C01778=1015.719,145.333,-122.552,166.904,54.935,160.108
C01779=1015.715,145.084,-122.532,166.901,54.946,160.110
C01780=1015.710,144.834,-122.514,166.899,54.957,160.111
C01781=1015.706,144.585,-122.494,166.895,54.967,160.113
C01782=1015.702,144.336,-122.475,166.892,54.977,160.114
C01783=1015.696,144.086,-122.456,166.888,54.988,160.115
C01784=1015.692,143.837,-122.437,166.885,54.998,160.116
C01785=1015.687,143.588,-122.418,166.881,55.009,160.118
C01786=1015.683,143.339,-122.399,166.879,55.020,160.119
C01787=1015.678,143.090,-122.380,166.875,55.030,160.121
C01788=1015.674,142.841,-122.360,166.871,55.041,160.122
C01789=1015.669,142.591,-122.342,166.868,55.051,160.123
C01790=1015.665,142.342,-122.323,166.865,55.061,160.125
C01791=1015.661,142.093,-122.303,166.862,55.072,160.126
C01792=1015.655,141.843,-122.285,166.858,55.082,160.127
C01793=1015.651,141.594,-122.265,166.856,55.093,160.129
C01794=1015.647,141.345,-122.247,166.853,55.104,160.130
C01795=1015.642,141.096,-122.228,166.848,55.114,160.131
C01796=1015.637,140.847,-122.208,166.845,55.125,160.133
C01797=1015.633,140.597,-122.189,166.842,55.135,160.134
C01798=1015.628,140.348,-122.171,166.839,55.145,160.136
C01799=1015.624,140.099,-122.152,166.836,55.156,160.137
C01800=1015.619,139.850,-122.133,166.832,55.166,160.138
C01801=1015.615,139.601,-122.113,166.829,55.176,160.140
C01802=1015.611,139.351,-122.095,166.827,55.188,160.141
C01803=1015.606,139.106,-122.076,166.823,55.197,160.142
C01804=1015.602,138.863,-122.057,166.820,55.208,160.144
C01805=1015.598,138.618,-122.039,166.817,55.218,160.145
C01806=1015.594,138.374,-122.021,166.813,55.228,160.146
C01807=1015.588,138.130,-122.002,166.810,55.239,160.148
C01808=1015.584,137.886,-121.984,166.807,55.249,160.149
C01809=1015.580,137.641,-121.965,166.804,55.259,160.150
C01810=1015.575,137.397,-121.946,166.801,55.270,160.152
C01811=1015.571,137.147,-121.927,166.798,55.280,160.153
C01812=1015.566,136.898,-121.909,166.795,55.291,160.155
C01813=1015.561,136.649,-121.890,166.791,55.301,160.156
C01814=1015.557,136.400,-121.872,166.788,55.311,160.157
C01815=1015.552,136.151,-121.853,166.785,55.322,160.159
C01816=1015.548,135.901,-121.834,166.781,55.332,160.160
C01817=1015.543,135.652,-121.816,166.778,55.344,160.161
C01818=1015.539,135.403,-121.796,166.775,55.354,160.163
C01819=1015.534,135.153,-121.778,166.772,55.364,160.164
C01820=1015.530,134.904,-121.759,166.769,55.375,160.165
C01821=1015.525,134.655,-121.740,166.766,55.385,160.167
C01822=1015.521,134.406,-121.723,166.763,55.396,160.168
C01823=1015.517,134.157,-121.704,166.760,55.406,160.170
C01824=1015.512,133.907,-121.686,166.757,55.417,160.171
C01825=1015.507,133.658,-121.666,166.753,55.428,160.172
C01826=1015.503,133.409,-121.648,166.750,55.438,160.174
C01827=1015.498,133.160,-121.630,166.747,55.449,160.175
C01828=1015.493,132.911,-121.610,166.744,55.459,160.176
C01829=1015.489,132.661,-121.592,166.741,55.470,160.178
C01830=1015.485,132.412,-121.574,166.737,55.480,160.179
C01831=1015.479,132.121,-121.552,166.734,55.492,160.181
C01832=1015.474,131.830,-121.531,166.730,55.505,160.183
C01833=1015.469,131.539,-121.509,166.727,55.517,160.184
C01834=1015.463,131.249,-121.487,166.723,55.529,160.186
C01835=1015.459,131.000,-121.469,166.719,55.540,160.187
C01836=1015.454,130.750,-121.451,166.717,55.551,160.189
C01837=1015.450,130.501,-121.432,166.714,55.561,160.190
C01838=1015.446,130.252,-121.414,166.711,55.572,160.191
C01839=1015.441,130.003,-121.395,166.708,55.582,160.193
C01840=1015.437,129.753,-121.376,166.705,55.592,160.194
C01841=1015.432,129.504,-121.358,166.702,55.603,160.195
C01842=1015.427,129.255,-121.340,166.698,55.613,160.197
C01843=1015.423,129.005,-121.321,166.695,55.624,160.198
C01844=1015.418,128.756,-121.303,166.693,55.635,160.200
C01845=1015.413,128.506,-121.285,166.690,55.645,160.201
C01846=1015.409,128.257,-121.267,166.687,55.656,160.203
C01847=1015.404,128.008,-121.249,166.683,55.667,160.204
C01848=1015.400,127.759,-121.231,166.680,55.677,160.205
C01849=1015.395,127.510,-121.213,166.677,55.688,160.207
C01850=1015.390,127.260,-121.195,166.674,55.699,160.208
C01851=1015.386,127.010,-121.177,166.671,55.709,160.210
C01852=1015.381,126.761,-121.159,166.668,55.720,160.211
C01853=1015.376,126.512,-121.141,166.666,55.731,160.213
C01854=1015.371,126.262,-121.123,166.663,55.741,160.214
C01855=1015.367,126.014,-121.105,166.658,55.752,160.215
C01856=1015.362,125.764,-121.087,166.655,55.763,160.217
C01857=1015.358,125.515,-121.068,166.652,55.773,160.218
C01858=1015.353,125.266,-121.050,166.649,55.783,160.219
C01859=1015.348,125.016,-121.032,166.647,55.795,160.221
C01860=1015.344,124.767,-121.015,166.644,55.805,160.222
C01861=1015.339,124.518,-120.997,166.641,55.816,160.224
C01862=1015.335,124.268,-120.979,166.638,55.826,160.225
C01863=1015.330,124.019,-120.961,166.635,55.837,160.226
C01864=1015.325,123.770,-120.942,166.632,55.847,160.228
C01865=1015.321,123.521,-120.925,166.629,55.857,160.229
C01866=1015.316,123.271,-120.907,166.626,55.869,160.231
C01867=1015.311,122.990,-120.887,166.623,55.880,160.232
C01868=1015.306,122.709,-120.866,166.619,55.892,160.234
C01869=1015.301,122.429,-120.846,166.617,55.904,160.236
C01870=1015.296,122.148,-120.825,166.612,55.916,160.237
C01871=1015.291,121.899,-120.808,166.609,55.927,160.238
C01872=1015.287,121.650,-120.789,166.606,55.937,160.240
C01873=1015.282,121.400,-120.772,166.603,55.948,160.241
C01874=1015.277,121.150,-120.754,166.600,55.958,160.242
C01875=1015.273,120.902,-120.736,166.597,55.969,160.244
C01876=1015.268,120.652,-120.718,166.594,55.979,160.245
C01877=1015.264,120.402,-120.700,166.591,55.990,160.247
C01878=1015.260,120.154,-120.683,166.589,56.001,160.248
C01879=1015.255,119.904,-120.664,166.587,56.011,160.250
C01880=1015.250,119.655,-120.646,166.584,56.022,160.251
C01881=1015.246,119.405,-120.629,166.581,56.032,160.253
C01882=1015.242,119.156,-120.611,166.578,56.043,160.254
C01883=1015.237,118.907,-120.593,166.575,56.053,160.255
C01884=1015.232,118.658,-120.575,166.572,56.064,160.257
C01885=1015.228,118.408,-120.558,166.569,56.074,160.258
C01886=1015.223,118.159,-120.540,166.566,56.085,160.260
C01887=1015.219,117.910,-120.521,166.563,56.095,160.261
C01888=1015.214,117.660,-120.504,166.560,56.106,160.262
C01889=1015.210,117.411,-120.486,166.557,56.116,160.264
C01890=1015.205,117.162,-120.468,166.555,56.127,160.265
C01891=1015.200,116.912,-120.450,166.551,56.137,160.266
C01892=1015.196,116.663,-120.433,166.548,56.147,160.268
C01893=1015.192,116.414,-120.415,166.545,56.158,160.269
C01894=1015.187,116.164,-120.396,166.542,56.168,160.271
C01895=1015.183,115.915,-120.379,166.540,56.178,160.272
C01896=1015.178,115.666,-120.361,166.538,56.189,160.274
C01897=1015.174,115.417,-120.344,166.535,56.199,160.275
C01898=1015.170,115.167,-120.326,166.532,56.210,160.276
C01899=1015.165,114.918,-120.308,166.529,56.220,160.278
C01900=1015.161,114.669,-120.291,166.526,56.231,160.279
C01901=1015.156,114.419,-120.273,166.523,56.242,160.281
C01902=1015.151,114.170,-120.254,166.520,56.252,160.282
C01903=1015.147,113.921,-120.237,166.518,56.262,160.283
C01904=1015.143,113.671,-120.219,166.515,56.272,160.285
C01905=1015.139,113.422,-120.202,166.512,56.283,160.286
C01906=1015.134,113.173,-120.184,166.509,56.293,160.287
C01907=1015.129,112.923,-120.166,166.506,56.304,160.289
C01908=1015.125,112.674,-120.149,166.503,56.314,160.290
C01909=1015.121,112.425,-120.130,166.500,56.325,160.292
C01910=1015.117,112.175,-120.113,166.498,56.334,160.293
C01911=1015.112,111.926,-120.095,166.495,56.345,160.294
C01912=1015.107,111.676,-120.078,166.492,56.355,160.296
C01913=1015.103,111.427,-120.060,166.490,56.366,160.297
C01914=1015.098,111.178,-120.043,166.487,56.377,160.299
C01915=1015.094,110.928,-120.026,166.484,56.387,160.300
C01916=1015.089,110.679,-120.008,166.481,56.398,160.301
C01917=1015.085,110.429,-119.990,166.478,56.408,160.303
C01918=1015.080,110.181,-119.973,166.475,56.419,160.304
C01919=1015.076,109.931,-119.956,166.472,56.429,160.306
C01920=1015.072,109.682,-119.939,166.471,56.440,160.307
C01921=1015.066,109.433,-119.921,166.468,56.450,160.309
C01922=1015.062,109.183,-119.904,166.465,56.461,160.310
C01923=1015.058,108.933,-119.887,166.462,56.471,160.312
C01924=1015.053,108.684,-119.870,166.459,56.482,160.313
C01925=1015.048,108.435,-119.852,166.456,56.492,160.314
C01926=1015.043,108.185,-119.835,166.454,56.503,160.316
C01927=1015.039,107.936,-119.818,166.451,56.514,160.317
C01928=1015.034,107.686,-119.801,166.448,56.524,160.319
C01929=1015.030,107.438,-119.783,166.445,56.535,160.320
C01930=1015.025,107.188,-119.767,166.442,56.545,160.321
C01931=1015.020,106.907,-119.747,166.439,56.557,160.323
C01932=1015.015,106.626,-119.728,166.436,56.569,160.325
C01933=1015.009,106.346,-119.708,166.434,56.581,160.327
C01934=1015.004,106.065,-119.689,166.431,56.593,160.328
C01935=1015.000,105.816,-119.672,166.428,56.603,160.329
C01936=1014.995,105.566,-119.655,166.425,56.614,160.331
C01937=1014.991,105.317,-119.638,166.422,56.625,160.332
C01938=1014.985,105.068,-119.621,166.419,56.634,160.333
C01939=1014.982,104.819,-119.604,166.416,56.645,160.335
C01940=1014.977,104.569,-119.586,166.413,56.656,160.336
C01941=1014.972,104.320,-119.570,166.411,56.666,160.338
C01942=1014.968,104.070,-119.552,166.409,56.676,160.339
C01943=1014.963,103.821,-119.536,166.406,56.687,160.341
C01944=1014.959,103.571,-119.518,166.403,56.698,160.342
C01945=1014.954,103.323,-119.501,166.401,56.708,160.344
C01946=1014.950,103.073,-119.484,166.398,56.719,160.345
C01947=1014.945,102.824,-119.467,166.395,56.729,160.346
C01948=1014.941,102.574,-119.450,166.392,56.740,160.348
C01949=1014.936,102.325,-119.433,166.390,56.750,160.349
C01950=1014.932,102.075,-119.416,166.387,56.760,160.351
C01951=1014.927,101.826,-119.399,166.385,56.771,160.352
C01952=1014.923,101.576,-119.382,166.382,56.782,160.354
C01953=1014.918,101.327,-119.366,166.378,56.792,160.355
C01954=1014.914,101.078,-119.348,166.377,56.802,160.356
C01955=1014.909,100.829,-119.332,166.374,56.812,160.358
C01956=1014.905,100.579,-119.315,166.371,56.823,160.359
C01957=1014.900,100.330,-119.298,166.368,56.833,160.360
C01958=1014.895,100.080,-119.280,166.365,56.844,160.362
C01959=1014.891,99.831,-119.263,166.364,56.854,160.363
C01960=1014.886,99.581,-119.246,166.361,56.864,160.365
C01961=1014.882,99.332,-119.229,166.358,56.874,160.366
C01962=1014.878,99.083,-119.212,166.355,56.885,160.367
C01963=1014.872,98.833,-119.196,166.353,56.895,160.369
C01964=1014.869,98.584,-119.179,166.350,56.906,160.370
C01965=1014.864,98.334,-119.162,166.348,56.917,160.372
C01966=1014.859,98.085,-119.146,166.345,56.927,160.373
C01967=1014.854,97.836,-119.129,166.342,56.938,160.375
C01968=1014.849,97.586,-119.112,166.339,56.948,160.376
C01969=1014.845,97.337,-119.095,166.336,56.959,160.377
C01970=1014.840,97.087,-119.079,166.335,56.969,160.379
C01971=1014.836,96.838,-119.063,166.332,56.979,160.381
C01972=1014.831,96.589,-119.046,166.329,56.990,160.382
C01973=1014.827,96.339,-119.029,166.327,57.001,160.383
C01974=1014.822,96.090,-119.012,166.323,57.011,160.385
C01975=1014.818,95.841,-118.996,166.321,57.021,160.386
C01976=1014.813,95.591,-118.980,166.319,57.032,160.388
C01977=1014.808,95.342,-118.963,166.316,57.042,160.389
C01978=1014.804,95.092,-118.946,166.314,57.053,160.391
C01979=1014.799,94.843,-118.929,166.310,57.063,160.392
C01980=1014.795,94.593,-118.914,166.308,57.074,160.393
C01981=1014.789,94.344,-118.897,166.306,57.084,160.395
C01982=1014.785,94.095,-118.880,166.303,57.095,160.396
C01983=1014.781,93.845,-118.863,166.300,57.105,160.397
C01984=1014.776,93.595,-118.847,166.298,57.115,160.399
C01985=1014.771,93.346,-118.831,166.296,57.126,160.401
C01986=1014.767,93.097,-118.814,166.293,57.136,160.402
C01987=1014.762,92.847,-118.797,166.290,57.146,160.403
C01988=1014.758,92.598,-118.781,166.287,57.157,160.405
C01989=1014.753,92.349,-118.764,166.286,57.167,160.406
C01990=1014.749,92.100,-118.748,166.283,57.177,160.407
C01991=1014.744,91.850,-118.731,166.280,57.188,160.409
C01992=1014.740,91.600,-118.715,166.277,57.199,160.410
C01993=1014.735,91.351,-118.698,166.275,57.208,160.412
C01994=1014.730,91.102,-118.681,166.273,57.219,160.413
C01995=1014.725,90.821,-118.663,166.269,57.231,160.415
C01996=1014.721,90.541,-118.645,166.267,57.242,160.416
C01997=1014.715,90.260,-118.626,166.264,57.254,160.418
C01998=1014.710,89.980,-118.608,166.261,57.265,160.419
C01999=1014.705,89.730,-118.591,166.259,57.275,160.421
C02000=1014.701,89.481,-118.574,166.256,57.286,160.422
C02001=1014.697,89.232,-118.558,166.253,57.296,160.424
C02002=1014.692,88.983,-118.542,166.252,57.306,160.425
C02003=1014.687,88.732,-118.526,166.249,57.316,160.426
C02004=1014.683,88.483,-118.509,166.246,57.327,160.428
C02005=1014.678,88.234,-118.493,166.243,57.338,160.429
C02006=1014.674,87.985,-118.477,166.241,57.347,160.431
C02007=1014.669,87.735,-118.461,166.239,57.358,160.432
C02008=1014.664,87.486,-118.444,166.236,57.369,160.434
C02009=1014.660,87.236,-118.428,166.233,57.380,160.435
C02010=1014.655,86.987,-118.412,166.231,57.389,160.437
C02011=1014.650,86.737,-118.396,166.229,57.400,160.438
C02012=1014.645,86.488,-118.380,166.226,57.411,160.439
C02013=1014.641,86.239,-118.364,166.223,57.421,160.441
C02014=1014.637,85.989,-118.348,166.222,57.431,160.442
C02015=1014.631,85.739,-118.332,166.219,57.442,160.444
C02016=1014.627,85.490,-118.316,166.216,57.452,160.445
C02017=1014.622,85.241,-118.299,166.213,57.463,160.446
C02018=1014.618,84.991,-118.284,166.212,57.473,160.448
C02019=1014.614,84.742,-118.268,166.209,57.483,160.449
C02020=1014.608,84.492,-118.252,166.206,57.494,160.451
C02021=1014.604,84.243,-118.236,166.204,57.503,160.452
C02022=1014.599,83.994,-118.219,166.201,57.514,160.454
C02023=1014.595,83.744,-118.203,166.199,57.525,160.455
C02024=1014.590,83.495,-118.188,166.197,57.534,160.456
C02025=1014.586,83.246,-118.171,166.194,57.545,160.458
C02026=1014.581,82.995,-118.155,166.191,57.555,160.459
C02027=1014.577,82.746,-118.139,166.189,57.566,160.461
C02028=1014.571,82.497,-118.123,166.186,57.575,160.462
C02029=1014.567,82.248,-118.108,166.184,57.586,160.464
C02030=1014.563,81.998,-118.092,166.182,57.596,160.465
C02031=1014.558,81.749,-118.075,166.179,57.607,160.466
C02032=1014.553,81.499,-118.059,166.176,57.617,160.468
C02033=1014.549,81.249,-118.044,166.175,57.627,160.469
C02034=1014.544,81.000,-118.027,166.172,57.637,160.470
C02035=1014.540,80.751,-118.011,166.169,57.648,160.472
C02036=1014.535,80.501,-117.995,166.167,57.657,160.473
C02037=1014.530,80.252,-117.980,166.165,57.668,160.475
C02038=1014.526,80.003,-117.964,166.163,57.678,160.476
C02039=1014.521,79.753,-117.948,166.159,57.688,160.477
C02040=1014.517,79.503,-117.932,166.157,57.699,160.479
C02041=1014.512,79.254,-117.915,166.155,57.708,160.480
C02042=1014.508,79.004,-117.900,166.152,57.719,160.482
C02043=1014.503,78.755,-117.884,166.150,57.729,160.483
C02044=1014.499,78.506,-117.867,166.147,57.739,160.484
C02045=1014.494,78.257,-117.852,166.146,57.749,160.486
C02046=1014.489,78.007,-117.836,166.143,57.759,160.487
C02047=1014.485,77.758,-117.821,166.141,57.769,160.489
C02048=1014.480,77.508,-117.804,166.138,57.780,160.490
C02049=1014.476,77.258,-117.788,166.135,57.790,160.491
C02050=1014.471,77.009,-117.772,166.133,57.799,160.493
C02051=1014.467,76.759,-117.757,166.131,57.810,160.494
C02052=1014.462,76.510,-117.741,166.129,57.820,160.496
C02053=1014.458,76.260,-117.726,166.126,57.831,160.497
C02054=1014.453,76.011,-117.709,166.124,57.840,160.499
C02055=1014.448,75.762,-117.694,166.121,57.850,160.500
C02056=1014.444,75.513,-117.678,166.119,57.861,160.501
C02057=1014.439,75.263,-117.662,166.117,57.871,160.503
C02058=1014.434,75.014,-117.647,166.114,57.882,160.504
C02059=1014.429,74.733,-117.630,166.112,57.892,160.506
C02060=1014.424,74.453,-117.613,166.109,57.904,160.507
C02061=1014.419,74.173,-117.595,166.107,57.915,160.509
C02062=1014.413,73.893,-117.577,166.104,57.927,160.510
C02063=1014.409,73.643,-117.562,166.102,57.937,160.512
C02064=1014.404,73.394,-117.546,166.099,57.947,160.513
C02065=1014.400,73.144,-117.531,166.096,57.958,160.514
C02066=1014.395,72.895,-117.515,166.094,57.967,160.516
C02067=1014.390,72.645,-117.500,166.091,57.978,160.517
C02068=1014.386,72.396,-117.484,166.090,57.988,160.519
C02069=1014.380,72.146,-117.468,166.087,57.998,160.520
C02070=1014.376,71.896,-117.453,166.085,58.008,160.521
C02071=1014.372,71.647,-117.437,166.083,58.019,160.523
C02072=1014.367,71.397,-117.422,166.081,58.028,160.524
C02073=1014.363,71.148,-117.406,166.078,58.038,160.526
C02074=1014.357,70.899,-117.391,166.076,58.048,160.527
C02075=1014.353,70.649,-117.375,166.073,58.059,160.529
C02076=1014.348,70.399,-117.361,166.071,58.068,160.530
C02077=1014.344,70.150,-117.345,166.068,58.079,160.531
C02078=1014.340,69.900,-117.329,166.066,58.088,160.533
C02079=1014.335,69.651,-117.314,166.063,58.098,160.534
C02080=1014.331,69.402,-117.298,166.062,58.109,160.535
C02081=1014.326,69.153,-117.283,166.059,58.119,160.537
C02082=1014.322,68.903,-117.267,166.057,58.129,160.538
C02083=1014.317,68.654,-117.252,166.054,58.139,160.539
C02084=1014.312,68.404,-117.237,166.052,58.148,160.541
C02085=1014.307,68.155,-117.221,166.050,58.159,160.542
C02086=1014.303,67.905,-117.206,166.048,58.169,160.544
C02087=1014.298,67.655,-117.191,166.046,58.179,160.545
C02088=1014.294,67.406,-117.175,166.043,58.189,160.546
C02089=1014.289,67.157,-117.160,166.041,58.198,160.548
C02090=1014.284,66.907,-117.145,166.038,58.209,160.549
C02091=1014.280,66.657,-117.130,166.037,58.219,160.551
C02092=1014.275,66.408,-117.115,166.034,58.229,160.552
C02093=1014.271,66.158,-117.099,166.032,58.239,160.553
C02094=1014.265,65.909,-117.084,166.029,58.249,160.555
C02095=1014.261,65.659,-117.069,166.027,58.259,160.556
C02096=1014.256,65.410,-117.054,166.024,58.269,160.557
C02097=1014.251,65.160,-117.038,166.022,58.279,160.559
C02098=1014.247,64.910,-117.023,166.020,58.289,160.560
C02099=1014.243,64.662,-117.009,166.018,58.299,160.562
C02100=1014.238,64.412,-116.993,166.016,58.309,160.563
C02101=1014.234,64.163,-116.978,166.013,58.319,160.564
C02102=1014.229,63.913,-116.963,166.011,58.329,160.566
C02103=1014.224,63.664,-116.948,166.008,58.339,160.567
C02104=1014.220,63.414,-116.932,166.007,58.349,160.568
C02105=1014.215,63.164,-116.918,166.004,58.359,160.570
C02106=1014.210,62.915,-116.903,166.002,58.368,160.571
C02107=1014.206,62.665,-116.888,166.000,58.378,160.572
C02108=1014.201,62.415,-116.872,165.997,58.388,160.574
C02109=1014.196,62.167,-116.858,165.995,58.398,160.575
C02110=1014.192,61.917,-116.843,165.993,58.409,160.577
C02111=1014.187,61.667,-116.829,165.991,58.419,160.578
C02112=1014.182,61.418,-116.813,165.988,58.429,160.579
C02113=1014.177,61.168,-116.799,165.986,58.439,160.581
C02114=1014.172,60.919,-116.784,165.983,58.449,160.582
C02115=1014.167,60.669,-116.769,165.981,58.458,160.583
C02116=1014.162,60.419,-116.754,165.979,58.469,160.585
C02117=1014.158,60.170,-116.740,165.977,58.479,160.586
C02118=1014.153,59.921,-116.725,165.974,58.489,160.588
C02119=1014.148,59.671,-116.710,165.973,58.499,160.589
C02120=1014.144,59.421,-116.696,165.970,58.509,160.590
C02121=1014.138,59.172,-116.681,165.968,58.519,160.592
C02122=1014.134,58.922,-116.666,165.966,58.529,160.593
C02123=1014.129,58.642,-116.649,165.963,58.540,160.595
C02124=1014.123,58.362,-116.633,165.961,58.551,160.596
C02125=1014.118,58.082,-116.617,165.958,58.562,160.598
C02126=1014.113,57.802,-116.600,165.955,58.573,160.599
C02127=1014.108,57.552,-116.585,165.953,58.583,160.600
C02128=1014.103,57.303,-116.570,165.951,58.593,160.602
C02129=1014.099,57.053,-116.556,165.948,58.603,160.603
C02130=1014.094,56.804,-116.542,165.947,58.613,160.605
C02131=1014.089,56.554,-116.527,165.944,58.623,160.606
C02132=1014.085,56.304,-116.512,165.942,58.633,160.607
C02133=1014.080,56.055,-116.498,165.940,58.642,160.609
C02134=1014.075,55.805,-116.482,165.937,58.653,160.610
C02135=1014.071,55.556,-116.468,165.936,58.662,160.611
C02136=1014.066,55.306,-116.454,165.934,58.672,160.613
C02137=1014.061,55.057,-116.439,165.931,58.682,160.614
C02138=1014.056,54.807,-116.424,165.928,58.691,160.615
C02139=1014.052,54.558,-116.410,165.927,58.701,160.617
C02140=1014.047,54.309,-116.395,165.924,58.711,160.618
C02141=1014.042,54.059,-116.381,165.922,58.721,160.619
C02142=1014.038,53.809,-116.366,165.920,58.731,160.621
C02143=1014.033,53.560,-116.351,165.918,58.740,160.622
C02144=1014.028,53.310,-116.337,165.915,58.750,160.623
C02145=1014.024,53.061,-116.322,165.913,58.760,160.625
C02146=1014.019,52.811,-116.307,165.912,58.770,160.626
C02147=1014.015,52.562,-116.293,165.910,58.779,160.628
C02148=1014.010,52.312,-116.279,165.906,58.789,160.629
C02149=1014.005,52.062,-116.264,165.905,58.799,160.630
C02150=1014.000,51.813,-116.249,165.903,58.808,160.632
C02151=1013.996,51.564,-116.235,165.900,58.817,160.633
C02152=1013.991,51.314,-116.220,165.898,58.828,160.634
C02153=1013.986,51.064,-116.206,165.896,58.837,160.635
C02154=1013.982,50.816,-116.191,165.894,58.847,160.637
C02155=1013.977,50.566,-116.177,165.892,58.856,160.638
C02156=1013.972,50.316,-116.162,165.890,58.866,160.640
C02157=1013.968,50.066,-116.148,165.888,58.875,160.641
C02158=1013.963,49.817,-116.133,165.885,58.885,160.642
C02159=1013.959,49.567,-116.119,165.883,58.894,160.643
C02160=1013.954,49.318,-116.104,165.881,58.904,160.645
C02161=1013.950,49.068,-116.090,165.878,58.913,160.646
C02162=1013.945,48.818,-116.076,165.877,58.923,160.647
C02163=1013.940,48.569,-116.060,165.875,58.933,160.649
C02164=1013.936,48.320,-116.046,165.873,58.942,160.650
C02165=1013.931,48.070,-116.032,165.870,58.952,160.651
C02166=1013.926,47.820,-116.017,165.868,58.961,160.652
C02167=1013.922,47.571,-116.003,165.866,58.971,160.654
C02168=1013.917,47.322,-115.988,165.863,58.980,160.655
C02169=1013.912,47.072,-115.974,165.861,58.989,160.656
C02170=1013.908,46.823,-115.960,165.859,58.999,160.657
C02171=1013.903,46.573,-115.945,165.857,59.008,160.659
C02172=1013.899,46.323,-115.931,165.855,59.018,160.660
C02173=1013.895,46.074,-115.917,165.853,59.027,160.661
C02174=1013.890,45.824,-115.901,165.851,59.036,160.662
C02175=1013.885,45.575,-115.887,165.849,59.046,160.664
C02176=1013.881,45.325,-115.873,165.847,59.055,160.665
C02177=1013.876,45.076,-115.858,165.845,59.065,160.667
C02178=1013.872,44.826,-115.844,165.843,59.074,160.668
C02179=1013.867,44.576,-115.830,165.840,59.083,160.669
C02180=1013.862,44.327,-115.815,165.839,59.093,160.670
C02181=1013.858,44.078,-115.801,165.836,59.102,160.671
C02182=1013.853,43.828,-115.786,165.834,59.111,160.673
C02183=1013.849,43.579,-115.772,165.832,59.120,160.674
C02184=1013.844,43.329,-115.758,165.830,59.130,160.675
C02185=1013.840,43.079,-115.743,165.828,59.139,160.676
C02186=1013.835,42.830,-115.729,165.825,59.148,160.678
C02187=1013.830,42.549,-115.713,165.823,59.158,160.679
C02188=1013.825,42.270,-115.696,165.821,59.169,160.680
C02189=1013.820,41.990,-115.680,165.819,59.179,160.682
C02190=1013.815,41.709,-115.665,165.816,59.189,160.683
C02191=1013.811,41.460,-115.650,165.814,59.198,160.684
C02192=1013.805,41.210,-115.637,165.812,59.208,160.686
C02193=1013.801,40.961,-115.622,165.810,59.217,160.687
C02194=1013.796,40.711,-115.608,165.808,59.226,160.688
C02195=1013.792,40.461,-115.595,165.806,59.236,160.690
C02196=1013.787,40.212,-115.581,165.804,59.245,160.691
C02197=1013.782,39.962,-115.566,165.802,59.254,160.692
C02198=1013.778,39.713,-115.552,165.799,59.263,160.693
C02199=1013.773,39.463,-115.538,165.798,59.273,160.695
C02200=1013.768,39.214,-115.524,165.795,59.282,160.696
C02201=1013.764,38.964,-115.510,165.793,59.292,160.697
C02202=1013.760,38.715,-115.496,165.791,59.301,160.698
C02203=1013.754,38.465,-115.483,165.789,59.310,160.699
C02204=1013.750,38.215,-115.468,165.787,59.320,160.701
C02205=1013.745,37.965,-115.454,165.785,59.329,160.702
C02206=1013.741,37.717,-115.441,165.782,59.338,160.703
C02207=1013.736,37.467,-115.426,165.780,59.347,160.704
C02208=1013.732,37.218,-115.412,165.778,59.356,160.706
C02209=1013.727,36.967,-115.399,165.776,59.365,160.707
C02210=1013.722,36.718,-115.385,165.774,59.374,160.708
C02211=1013.718,36.468,-115.370,165.772,59.383,160.709
C02212=1013.713,36.218,-115.356,165.770,59.392,160.710
C02213=1013.708,35.969,-115.343,165.768,59.401,160.712
C02214=1013.704,35.719,-115.329,165.766,59.411,160.713
C02215=1013.699,35.470,-115.315,165.764,59.420,160.714
C02216=1013.694,35.220,-115.302,165.762,59.429,160.716
C02217=1013.689,34.971,-115.288,165.759,59.438,160.717
C02218=1013.685,34.722,-115.274,165.757,59.447,160.718
C02219=1013.680,34.471,-115.261,165.755,59.457,160.719
C02220=1013.675,34.223,-115.247,165.753,59.466,160.720
C02221=1013.671,33.972,-115.233,165.750,59.475,160.721
C02222=1013.666,33.723,-115.220,165.749,59.484,160.723
C02223=1013.661,33.473,-115.205,165.748,59.493,160.724
C02224=1013.657,33.224,-115.193,165.745,59.502,160.726
C02225=1013.652,32.974,-115.178,165.743,59.512,160.727
C02226=1013.647,32.724,-115.165,165.741,59.521,160.728
C02227=1013.642,32.475,-115.151,165.739,59.530,160.729
C02228=1013.638,32.226,-115.137,165.737,59.539,160.730
C02229=1013.633,31.976,-115.125,165.735,59.547,160.731
C02230=1013.628,31.726,-115.110,165.733,59.556,160.732
C02231=1013.624,31.477,-115.097,165.730,59.565,160.734
C02232=1013.619,31.227,-115.083,165.728,59.574,160.735
C02233=1013.615,30.977,-115.070,165.726,59.584,160.736
C02234=1013.610,30.727,-115.056,165.725,59.592,160.737
C02235=1013.605,30.478,-115.043,165.723,59.601,160.739
C02236=1013.600,30.229,-115.029,165.720,59.610,160.740
C02237=1013.596,29.979,-115.015,165.718,59.620,160.741
C02238=1013.591,29.730,-115.002,165.716,59.628,160.742
C02239=1013.586,29.480,-114.988,165.714,59.637,160.743
C02240=1013.582,29.230,-114.975,165.712,59.646,160.744
C02241=1013.578,28.981,-114.961,165.710,59.655,160.746
C02242=1013.572,28.731,-114.948,165.709,59.664,160.747
C02243=1013.568,28.482,-114.934,165.706,59.672,160.748
C02244=1013.563,28.232,-114.920,165.704,59.681,160.749
C02245=1013.558,27.983,-114.907,165.703,59.690,160.750
C02246=1013.554,27.733,-114.894,165.700,59.698,160.751
C02247=1013.549,27.483,-114.880,165.698,59.708,160.753
C02248=1013.545,27.234,-114.866,165.696,59.716,160.754
C02249=1013.540,26.983,-114.853,165.694,59.725,160.755
C02250=1013.535,26.734,-114.840,165.691,59.734,160.756
C02251=1013.530,26.454,-114.825,165.690,59.744,160.758
C02252=1013.525,26.174,-114.810,165.687,59.754,160.759
C02253=1013.520,25.894,-114.794,165.685,59.763,160.760
C02254=1013.515,25.615,-114.780,165.683,59.774,160.761
C02255=1013.509,25.365,-114.766,165.680,59.783,160.763
C02256=1013.505,25.115,-114.754,165.679,59.791,160.764
C02257=1013.501,24.866,-114.740,165.677,59.800,160.765
C02258=1013.496,24.616,-114.726,165.674,59.809,160.766
C02259=1013.491,24.367,-114.714,165.673,59.817,160.767
C02260=1013.486,24.117,-114.701,165.670,59.826,160.768
C02261=1013.481,23.867,-114.688,165.668,59.835,160.769
C02262=1013.477,23.618,-114.674,165.667,59.843,160.771
C02263=1013.473,23.368,-114.661,165.664,59.853,160.772
C02264=1013.467,23.118,-114.648,165.662,59.861,160.773
C02265=1013.462,22.869,-114.634,165.661,59.870,160.774
C02266=1013.458,22.620,-114.621,165.658,59.878,160.775
C02267=1013.453,22.369,-114.608,165.657,59.887,160.776
C02268=1013.449,22.120,-114.595,165.654,59.895,160.777
C02269=1013.444,21.870,-114.582,165.653,59.904,160.779
C02270=1013.439,21.621,-114.569,165.650,59.912,160.779
C02271=1013.434,21.371,-114.555,165.648,59.922,160.781
C02272=1013.430,21.122,-114.543,165.646,59.930,160.782
C02273=1013.426,20.872,-114.529,165.644,59.939,160.783
C02274=1013.421,20.623,-114.516,165.642,59.947,160.784
C02275=1013.416,20.373,-114.503,165.639,59.955,160.785
C02276=1013.411,20.123,-114.490,165.638,59.964,160.786
C02277=1013.407,19.874,-114.477,165.636,59.972,160.787
C02278=1013.402,19.623,-114.463,165.635,59.981,160.789
C02279=1013.397,19.374,-114.450,165.632,59.990,160.790
C02280=1013.393,19.125,-114.437,165.630,59.998,160.791
C02281=1013.388,18.875,-114.424,165.628,60.007,160.792
C02282=1013.383,18.625,-114.411,165.626,60.015,160.793
C02283=1013.379,18.376,-114.398,165.623,60.023,160.794
C02284=1013.374,18.126,-114.386,165.622,60.032,160.795
C02285=1013.370,17.876,-114.372,165.620,60.040,160.796
C02286=1013.365,17.626,-114.359,165.618,60.048,160.797
C02287=1013.360,17.377,-114.346,165.615,60.057,160.798
C02288=1013.356,17.127,-114.333,165.614,60.066,160.799
C02289=1013.351,16.878,-114.321,165.612,60.074,160.801
C02290=1013.347,16.628,-114.308,165.610,60.082,160.801
C02291=1013.342,16.378,-114.295,165.608,60.090,160.802
C02292=1013.337,16.129,-114.282,165.606,60.099,160.804
C02293=1013.332,15.880,-114.268,165.604,60.107,160.805
C02294=1013.328,15.630,-114.256,165.601,60.116,160.806
C02295=1013.323,15.381,-114.243,165.600,60.124,160.807
C02296=1013.318,15.131,-114.230,165.598,60.132,160.808
C02297=1013.313,14.881,-114.217,165.596,60.141,160.809
C02298=1013.309,14.632,-114.204,165.594,60.149,160.810
C02299=1013.304,14.382,-114.191,165.593,60.157,160.811
C02300=1013.300,14.133,-114.179,165.590,60.165,160.812
C02301=1013.295,13.883,-114.166,165.588,60.173,160.813
C02302=1013.290,13.633,-114.153,165.587,60.181,160.814
C02303=1013.286,13.383,-114.141,165.584,60.190,160.815
C02304=1013.281,13.133,-114.128,165.582,60.198,160.816
C02305=1013.276,12.884,-114.115,165.580,60.206,160.817
C02306=1013.272,12.634,-114.102,165.578,60.214,160.818
C02307=1013.267,12.384,-114.089,165.576,60.222,160.819
C02308=1013.261,12.135,-114.077,165.574,60.230,160.820
C02309=1013.257,11.885,-114.065,165.572,60.240,160.822
C02310=1013.252,11.635,-114.052,165.571,60.248,160.823
C02311=1013.248,11.386,-114.039,165.568,60.256,160.824
C02312=1013.243,11.137,-114.027,165.566,60.264,160.825
C02313=1013.238,10.887,-114.014,165.565,60.272,160.826
C02314=1013.234,10.637,-114.002,165.562,60.281,160.827
C02315=1013.228,10.358,-113.988,165.560,60.290,160.828
C02316=1013.223,10.080,-113.975,165.557,60.298,160.829
C02317=1013.218,9.801,-113.960,165.555,60.308,160.830
C02318=1013.212,9.523,-113.946,165.553,60.317,160.831
C02319=1013.208,9.274,-113.933,165.551,60.325,160.832
C02320=1013.203,9.024,-113.922,165.550,60.333,160.833
C02321=1013.198,8.774,-113.909,165.548,60.341,160.835
C02322=1013.193,8.524,-113.896,165.545,60.349,160.835
C02323=1013.189,8.274,-113.884,165.543,60.357,160.836
C02324=1013.183,8.025,-113.872,165.541,60.365,160.837
C02325=1013.179,7.776,-113.859,165.540,60.373,160.838
C02326=1013.174,7.526,-113.846,165.538,60.381,160.840
C02327=1013.170,7.276,-113.834,165.535,60.389,160.840
C02328=1013.165,7.027,-113.822,165.533,60.397,160.841
C02329=1013.160,6.777,-113.809,165.531,60.405,160.842
C02330=1013.156,6.527,-113.797,165.530,60.413,160.843
C02331=1013.151,6.278,-113.784,165.528,60.421,160.844
C02332=1013.146,6.029,-113.772,165.526,60.428,160.845
C02333=1013.142,5.779,-113.760,165.524,60.436,160.846
C02334=1013.137,5.529,-113.747,165.521,60.445,160.847
C02335=1013.132,5.280,-113.735,165.519,60.452,160.848
C02336=1013.128,5.030,-113.723,165.518,60.460,160.849
C02337=1013.123,4.780,-113.710,165.516,60.468,160.850
C02338=1013.119,4.530,-113.698,165.514,60.475,160.851
C02339=1013.113,4.281,-113.686,165.512,60.483,160.852
C02340=1013.109,4.031,-113.673,165.510,60.491,160.853
C02341=1013.105,3.781,-113.661,165.508,60.499,160.854
C02342=1013.100,3.532,-113.648,165.506,60.506,160.855
C02343=1013.095,3.283,-113.636,165.504,60.514,160.856
C02344=1013.090,3.033,-113.624,165.502,60.521,160.857
C02345=1013.086,2.783,-113.611,165.500,60.529,160.858
C02346=1013.082,2.533,-113.599,165.498,60.537,160.858
C02347=1013.076,2.284,-113.587,165.496,60.545,160.860
C02348=1013.072,2.034,-113.574,165.494,60.552,160.860
C02349=1013.067,1.784,-113.562,165.492,60.560,160.861
C02350=1013.062,1.535,-113.550,165.490,60.567,160.862
C02351=1013.058,1.285,-113.538,165.488,60.575,160.863
C02352=1013.053,1.035,-113.525,165.486,60.583,160.864
C02353=1013.049,0.785,-113.513,165.484,60.590,160.865
C02354=1013.044,0.536,-113.501,165.483,60.597,160.866
C02355=1013.039,0.287,-113.488,165.481,60.605,160.867
C02356=1013.035,0.036,-113.476,165.479,60.612,160.868
C02357=1013.030,-0.213,-113.463,165.477,60.619,160.868
C02358=1013.025,-0.463,-113.452,165.474,60.627,160.869
C02359=1013.021,-0.712,-113.439,165.473,60.635,160.870
C02360=1013.017,-0.962,-113.427,165.470,60.642,160.871
C02361=1013.011,-1.212,-113.415,165.469,60.649,160.872
C02362=1013.007,-1.462,-113.403,165.467,60.656,160.873
C02363=1013.002,-1.711,-113.390,165.465,60.664,160.874
C02364=1012.998,-1.961,-113.378,165.463,60.672,160.875
C02365=1012.993,-2.210,-113.366,165.462,60.679,160.876
C02366=1012.989,-2.461,-113.354,165.460,60.686,160.876
C02367=1012.985,-2.709,-113.341,165.457,60.693,160.877
C02368=1012.980,-2.959,-113.330,165.455,60.700,160.878
C02369=1012.975,-3.209,-113.317,165.454,60.707,160.879
C02370=1012.971,-3.459,-113.305,165.452,60.715,160.880
C02371=1012.966,-3.708,-113.292,165.449,60.722,160.880
C02372=1012.961,-3.958,-113.281,165.447,60.729,160.881
C02373=1012.957,-4.208,-113.268,165.446,60.736,160.882
C02374=1012.952,-4.458,-113.256,165.444,60.743,160.883
C02375=1012.948,-4.708,-113.244,165.441,60.751,160.884
C02376=1012.943,-4.957,-113.232,165.440,60.758,160.885
C02377=1012.938,-5.206,-113.220,165.438,60.765,160.885
C02378=1012.934,-5.456,-113.208,165.436,60.772,160.886
C02379=1012.928,-5.748,-113.194,165.433,60.781,160.887
C02380=1012.923,-6.040,-113.181,165.431,60.789,160.888
C02381=1012.918,-6.330,-113.167,165.429,60.798,160.890
C02382=1012.912,-6.622,-113.153,165.427,60.807,160.890
C02383=1012.907,-6.871,-113.142,165.425,60.813,160.891
C02384=1012.902,-7.121,-113.130,165.423,60.820,160.892
C02385=1012.897,-7.371,-113.118,165.420,60.828,160.893
C02386=1012.893,-7.620,-113.107,165.419,60.834,160.894
C02387=1012.888,-7.870,-113.095,165.417,60.842,160.894
C02388=1012.883,-8.120,-113.083,165.415,60.849,160.895
C02389=1012.878,-8.369,-113.072,165.414,60.856,160.896
C02390=1012.874,-8.620,-113.060,165.411,60.863,160.897
C02391=1012.869,-8.869,-113.048,165.409,60.871,160.898
C02392=1012.864,-9.118,-113.036,165.408,60.877,160.899
C02393=1012.860,-9.368,-113.024,165.405,60.884,160.899
C02394=1012.855,-9.618,-113.013,165.404,60.891,160.900
C02395=1012.850,-9.868,-113.001,165.402,60.898,160.901
C02396=1012.846,-10.118,-112.989,165.400,60.905,160.902
C02397=1012.842,-10.367,-112.978,165.397,60.912,160.902
C02398=1012.837,-10.617,-112.967,165.395,60.919,160.903
C02399=1012.830,1.156,-113.950,165.465,60.816,160.904
C02400=1012.834,1.406,-113.963,165.466,60.809,160.903
C02401=1012.839,1.656,-113.974,165.468,60.801,160.903
C02402=1012.844,1.905,-113.987,165.470,60.794,160.902
C02403=1012.848,2.155,-113.999,165.471,60.786,160.900
C02404=1012.853,2.404,-114.011,165.473,60.779,160.900
C02405=1012.857,2.654,-114.023,165.475,60.772,160.899
C02406=1012.862,2.903,-114.036,165.478,60.764,160.898
C02407=1012.866,3.154,-114.048,165.479,60.758,160.897
C02408=1012.871,3.403,-114.060,165.481,60.750,160.896
C02409=1012.876,3.652,-114.073,165.483,60.743,160.896
C02410=1012.880,3.902,-114.085,165.485,60.735,160.894
C02411=1012.885,4.152,-114.097,165.487,60.728,160.894
C02412=1012.890,4.402,-114.109,165.488,60.721,160.893
C02413=1012.894,4.651,-114.122,165.490,60.713,160.892
C02414=1012.899,4.901,-114.134,165.492,60.705,160.891
C02415=1012.904,5.150,-114.146,165.494,60.698,160.890
C02416=1012.909,5.400,-114.159,165.497,60.691,160.889
C02417=1012.913,5.650,-114.171,165.498,60.683,160.888
C02418=1012.917,5.900,-114.184,165.501,60.675,160.887
C02419=1012.922,6.149,-114.195,165.502,60.667,160.886
C02420=1012.927,6.399,-114.208,165.504,60.660,160.885
C02421=1012.931,6.648,-114.221,165.506,60.653,160.884
C02422=1012.936,6.898,-114.233,165.507,60.645,160.883
C02423=1012.941,7.148,-114.245,165.509,60.638,160.883
C02424=1012.946,7.397,-114.258,165.511,60.630,160.881
C02425=1012.950,7.647,-114.270,165.513,60.622,160.881
C02426=1012.954,7.897,-114.282,165.515,60.614,160.880
C02427=1012.959,8.147,-114.294,165.517,60.607,160.879
C02428=1012.964,8.396,-114.307,165.519,60.599,160.878
C02429=1012.969,8.645,-114.320,165.521,60.592,160.877
C02430=1012.974,8.895,-114.331,165.523,60.584,160.876
C02431=1012.978,9.145,-114.344,165.524,60.576,160.875
C02432=1012.985,9.510,-114.362,165.528,60.565,160.874
C02433=1012.992,9.875,-114.380,165.530,60.553,160.872
C02434=1012.999,10.240,-114.398,165.533,60.541,160.871
C02435=1013.006,10.606,-114.417,165.536,60.529,160.869
C02436=1013.010,10.855,-114.429,165.538,60.522,160.868
C02437=1013.015,11.105,-114.442,165.540,60.514,160.867
C02438=1013.020,11.354,-114.454,165.541,60.506,160.866
C02439=1013.025,11.604,-114.466,165.544,60.498,160.865
C02440=1013.029,11.853,-114.479,165.546,60.490,160.864
C02441=1013.034,12.103,-114.492,165.548,60.482,160.863
C02442=1013.039,12.353,-114.503,165.550,60.474,160.862
C02443=1013.043,12.602,-114.516,165.551,60.466,160.861
C02444=1013.048,12.852,-114.529,165.554,60.458,160.860
C02445=1013.052,13.101,-114.542,165.555,60.450,160.859
C02446=1013.058,13.351,-114.555,165.558,60.442,160.858
C02447=1013.062,13.601,-114.568,165.559,60.434,160.857
C02448=1013.066,13.851,-114.580,165.561,60.426,160.856
C02449=1013.071,14.100,-114.593,165.563,60.418,160.855
C02450=1013.076,14.350,-114.605,165.564,60.410,160.854
C02451=1013.080,14.599,-114.618,165.568,60.402,160.853
C02452=1013.085,14.849,-114.631,165.569,60.394,160.852
C02453=1013.090,15.099,-114.644,165.571,60.386,160.851
C02454=1013.094,15.349,-114.657,165.573,60.378,160.850
C02455=1013.099,15.598,-114.670,165.574,60.370,160.849
C02456=1013.104,15.848,-114.682,165.577,60.362,160.848
C02457=1013.108,16.097,-114.695,165.578,60.354,160.847
C02458=1013.113,16.347,-114.708,165.580,60.346,160.846
C02459=1013.118,16.597,-114.721,165.582,60.338,160.845
C02460=1013.122,16.846,-114.734,165.584,60.329,160.844
C02461=1013.127,17.096,-114.747,165.586,60.321,160.843
C02462=1013.132,17.345,-114.759,165.588,60.313,160.841
C02463=1013.136,17.595,-114.772,165.589,60.305,160.840
C02464=1013.141,17.844,-114.785,165.592,60.297,160.839
C02465=1013.146,18.094,-114.798,165.594,60.289,160.838
C02466=1013.150,18.344,-114.812,165.595,60.281,160.837
C02467=1013.154,18.594,-114.824,165.598,60.272,160.836
C02468=1013.159,18.843,-114.837,165.600,60.264,160.835
C02469=1013.163,19.093,-114.850,165.601,60.256,160.834
C02470=1013.169,19.343,-114.863,165.604,60.248,160.833
C02471=1013.173,19.592,-114.876,165.605,60.239,160.832
C02472=1013.177,19.842,-114.889,165.607,60.231,160.831
C02473=1013.182,20.091,-114.903,165.610,60.222,160.830
C02474=1013.186,20.341,-114.915,165.611,60.214,160.829
C02475=1013.192,20.591,-114.929,165.613,60.206,160.828
C02476=1013.196,20.840,-114.941,165.616,60.198,160.827
C02477=1013.201,21.090,-114.954,165.617,60.190,160.826
C02478=1013.205,21.339,-114.968,165.619,60.181,160.824
C02479=1013.210,21.590,-114.981,165.621,60.173,160.823
C02480=1013.215,21.839,-114.994,165.623,60.165,160.822
C02481=1013.219,22.088,-115.007,165.625,60.156,160.821
C02482=1013.224,22.338,-115.020,165.626,60.147,160.820
C02483=1013.228,22.588,-115.034,165.629,60.139,160.819
C02484=1013.233,22.838,-115.046,165.631,60.131,160.818
C02485=1013.238,23.086,-115.060,165.633,60.122,160.817
C02486=1013.242,23.336,-115.073,165.635,60.114,160.816
C02487=1013.247,23.586,-115.086,165.637,60.105,160.815
C02488=1013.251,23.836,-115.099,165.638,60.097,160.813
C02489=1013.256,24.085,-115.112,165.641,60.088,160.812
C02490=1013.261,24.334,-115.125,165.642,60.079,160.811
C02491=1013.266,24.584,-115.139,165.645,60.071,160.810
C02492=1013.270,24.834,-115.151,165.647,60.063,160.809
C02493=1013.274,25.084,-115.165,165.649,60.054,160.808
C02494=1013.280,25.333,-115.179,165.650,60.046,160.807
C02495=1013.284,25.583,-115.191,165.653,60.037,160.805
C02496=1013.290,25.863,-115.206,165.655,60.027,160.804
C02497=1013.294,26.142,-115.221,165.657,60.017,160.803
C02498=1013.300,26.422,-115.236,165.659,60.008,160.802
C02499=1013.306,26.702,-115.251,165.661,59.999,160.800
C02500=1013.309,26.952,-115.264,165.663,59.989,160.799
C02501=1013.314,27.201,-115.277,165.664,59.981,160.798
C02502=1013.319,27.451,-115.291,165.667,59.972,160.797
C02503=1013.323,27.700,-115.304,165.669,59.963,160.796
C02504=1013.328,27.950,-115.317,165.671,59.955,160.795
C02505=1013.333,28.200,-115.332,165.673,59.946,160.793
C02506=1013.337,28.449,-115.344,165.675,59.938,160.792
C02507=1013.341,28.699,-115.358,165.677,59.929,160.791
C02508=1013.346,28.949,-115.372,165.679,59.921,160.790
C02509=1013.351,29.198,-115.385,165.681,59.912,160.789
C02510=1013.355,29.447,-115.398,165.684,59.903,160.788
C02511=1013.361,29.697,-115.412,165.685,59.894,160.787
C02512=1013.364,29.947,-115.426,165.687,59.885,160.785
C02513=1013.369,30.196,-115.438,165.690,59.877,160.784
C02514=1013.374,30.446,-115.453,165.691,59.868,160.783
C02515=1013.378,30.696,-115.466,165.693,59.859,160.782
C02516=1013.382,30.945,-115.480,165.696,59.850,160.781
C02517=1013.388,31.195,-115.493,165.697,59.842,160.779
C02518=1013.393,31.444,-115.506,165.699,59.833,160.778
C02519=1013.397,31.694,-115.520,165.701,59.823,160.777
C02520=1013.402,31.943,-115.534,165.703,59.815,160.776
C02521=1013.406,32.193,-115.547,165.705,59.806,160.775
C02522=1013.411,32.443,-115.561,165.707,59.797,160.774
C02523=1013.415,32.692,-115.574,165.709,59.788,160.772
C02524=1013.420,32.942,-115.588,165.710,59.779,160.771
C02525=1013.425,33.191,-115.602,165.713,59.771,160.770
C02526=1013.429,33.441,-115.615,165.715,59.762,160.769
C02527=1013.435,33.690,-115.629,165.717,59.752,160.768
C02528=1013.438,33.940,-115.642,165.719,59.744,160.766
C02529=1013.444,34.190,-115.656,165.721,59.735,160.765
C02530=1013.448,34.439,-115.669,165.723,59.725,160.764
C02531=1013.453,34.688,-115.683,165.725,59.716,160.763
C02532=1013.457,34.939,-115.697,165.727,59.707,160.761
C02533=1013.462,35.188,-115.710,165.729,59.698,160.760
C02534=1013.467,35.438,-115.725,165.730,59.689,160.759
C02535=1013.471,35.687,-115.737,165.733,59.680,160.758
C02536=1013.476,35.937,-115.752,165.735,59.671,160.756
C02537=1013.481,36.187,-115.765,165.737,59.662,160.755
C02538=1013.485,36.436,-115.779,165.739,59.653,160.754
C02539=1013.490,36.685,-115.793,165.741,59.645,160.753
C02540=1013.495,36.936,-115.806,165.743,59.636,160.752
C02541=1013.499,37.185,-115.821,165.745,59.626,160.751
C02542=1013.503,37.434,-115.835,165.748,59.617,160.749
C02543=1013.508,37.684,-115.848,165.750,59.608,160.748
C02544=1013.512,37.934,-115.862,165.752,59.599,160.747
C02545=1013.517,38.183,-115.876,165.753,59.590,160.746
C02546=1013.522,38.432,-115.890,165.755,59.581,160.744
C02547=1013.527,38.682,-115.904,165.757,59.572,160.743
C02548=1013.531,38.931,-115.918,165.760,59.563,160.742
C02549=1013.536,39.182,-115.932,165.762,59.554,160.741
C02550=1013.540,39.431,-115.946,165.764,59.545,160.740
C02551=1013.545,39.681,-115.960,165.766,59.535,160.738
C02552=1013.549,39.930,-115.974,165.767,59.526,160.737
C02553=1013.554,40.179,-115.988,165.769,59.517,160.736
C02554=1013.558,40.429,-116.001,165.771,59.508,160.734
C02555=1013.563,40.679,-116.016,165.773,59.499,160.733
C02556=1013.568,40.928,-116.029,165.776,59.490,160.732
C02557=1013.572,41.178,-116.044,165.778,59.480,160.731
C02558=1013.577,41.427,-116.058,165.780,59.471,160.730
C02559=1013.581,41.678,-116.072,165.782,59.461,160.728
C02560=1013.587,41.957,-116.087,165.784,59.451,160.727
C02561=1013.591,42.237,-116.104,165.787,59.441,160.725
C02562=1013.596,42.517,-116.119,165.789,59.431,160.724
C02563=1013.602,42.797,-116.136,165.791,59.421,160.723
C02564=1013.606,43.046,-116.150,165.793,59.412,160.721
C02565=1013.611,43.296,-116.164,165.796,59.402,160.720
C02566=1013.615,43.545,-116.178,165.798,59.393,160.719
C02567=1013.620,43.795,-116.193,165.800,59.383,160.718
C02568=1013.624,44.044,-116.207,165.801,59.375,160.716
C02569=1013.629,44.294,-116.221,165.803,59.366,160.715
C02570=1013.633,44.543,-116.236,165.805,59.357,160.714
C02571=1013.638,44.793,-116.250,165.807,59.347,160.713
C02572=1013.642,45.043,-116.265,165.810,59.338,160.712
C02573=1013.647,45.292,-116.279,165.811,59.328,160.710
C02574=1013.651,45.542,-116.293,165.814,59.319,160.709
C02575=1013.655,45.791,-116.307,165.816,59.310,160.708
C02576=1013.660,46.041,-116.322,165.818,59.301,160.706
C02577=1013.664,46.290,-116.336,165.820,59.291,160.705
C02578=1013.669,46.540,-116.350,165.822,59.282,160.704
C02579=1013.674,46.790,-116.365,165.824,59.273,160.703
C02580=1013.678,47.039,-116.379,165.826,59.263,160.701
C02581=1013.683,47.289,-116.394,165.828,59.254,160.700
C02582=1013.687,47.538,-116.408,165.830,59.245,160.699
C02583=1013.692,47.788,-116.422,165.832,59.235,160.697
C02584=1013.697,48.038,-116.437,165.834,59.226,160.696
C02585=1013.701,48.287,-116.451,165.836,59.216,160.695
C02586=1013.705,48.537,-116.465,165.838,59.207,160.693
C02587=1013.711,48.786,-116.481,165.841,59.198,160.692
C02588=1013.715,49.035,-116.495,165.842,59.188,160.691
C02589=1013.719,49.285,-116.509,165.846,59.179,160.690
C02590=1013.724,49.534,-116.523,165.847,59.169,160.688
C02591=1013.728,49.784,-116.538,165.850,59.160,160.687
C02592=1013.733,50.034,-116.552,165.851,59.150,160.686
C02593=1013.737,50.283,-116.566,165.853,59.141,160.684
C02594=1013.742,50.532,-116.581,165.855,59.131,160.683
C02595=1013.747,50.782,-116.596,165.857,59.122,160.682
C02596=1013.751,51.032,-116.610,165.859,59.112,160.680
C02597=1013.756,51.281,-116.624,165.862,59.103,160.679
C02598=1013.761,51.531,-116.639,165.864,59.093,160.678
C02599=1013.765,51.780,-116.654,165.866,59.084,160.677
C02600=1013.770,52.030,-116.668,165.868,59.074,160.675
C02601=1013.774,52.280,-116.683,165.870,59.064,160.674
C02602=1013.779,52.529,-116.697,165.873,59.055,160.673
C02603=1013.783,52.779,-116.711,165.875,59.045,160.671
C02604=1013.788,53.028,-116.726,165.877,59.035,160.670
C02605=1013.793,53.277,-116.740,165.879,59.026,160.669
C02606=1013.797,53.527,-116.756,165.881,59.016,160.667
C02607=1013.801,53.777,-116.770,165.883,59.006,160.666
C02608=1013.806,54.027,-116.785,165.886,58.997,160.665
C02609=1013.810,54.276,-116.799,165.887,58.987,160.663
C02610=1013.815,54.526,-116.814,165.889,58.977,160.662
C02611=1013.820,54.775,-116.828,165.892,58.967,160.660
C02612=1013.824,55.024,-116.843,165.894,58.958,160.659
C02613=1013.829,55.274,-116.857,165.896,58.948,160.658
C02614=1013.834,55.524,-116.872,165.899,58.938,160.657
C02615=1013.839,55.774,-116.886,165.900,58.928,160.655
C02616=1013.843,56.022,-116.901,165.902,58.918,160.654
C02617=1013.848,56.272,-116.916,165.904,58.909,160.652
C02618=1013.852,56.522,-116.930,165.907,58.899,160.651
C02619=1013.857,56.771,-116.944,165.909,58.889,160.650
C02620=1013.862,57.020,-116.959,165.911,58.879,160.648
C02621=1013.866,57.270,-116.974,165.913,58.869,160.647
C02622=1013.871,57.520,-116.988,165.915,58.859,160.646
C02623=1013.876,57.769,-117.003,165.918,58.849,160.644
C02624=1013.881,58.050,-117.019,165.920,58.838,160.643
C02625=1013.886,58.329,-117.035,165.922,58.827,160.641
C02626=1013.892,58.609,-117.053,165.924,58.816,160.639
C02627=1013.897,58.889,-117.068,165.928,58.805,160.638
C02628=1013.902,59.139,-117.083,165.929,58.795,160.637
C02629=1013.906,59.388,-117.098,165.932,58.785,160.635
C02630=1013.911,59.638,-117.112,165.934,58.775,160.634
C02631=1013.916,59.887,-117.127,165.936,58.765,160.632
C02632=1013.920,60.137,-117.142,165.939,58.755,160.631
C02633=1013.925,60.387,-117.156,165.940,58.745,160.630
C02634=1013.930,60.636,-117.171,165.943,58.735,160.628
C02635=1013.935,60.886,-117.186,165.945,58.725,160.627
C02636=1013.939,61.134,-117.200,165.948,58.715,160.626
C02637=1013.944,61.384,-117.215,165.950,58.705,160.624
C02638=1013.949,61.634,-117.229,165.952,58.695,160.623
C02639=1013.954,61.883,-117.245,165.954,58.686,160.622
C02640=1013.959,62.133,-117.259,165.957,58.675,160.620
C02641=1013.964,62.383,-117.274,165.959,58.666,160.619
C02642=1013.968,62.632,-117.288,165.961,58.655,160.617
C02643=1013.972,62.881,-117.304,165.963,58.646,160.616
C02644=1013.977,63.131,-117.319,165.965,58.636,160.615
C02645=1013.982,63.381,-117.334,165.968,58.626,160.613
C02646=1013.986,63.631,-117.349,165.970,58.616,160.612
C02647=1013.991,63.880,-117.364,165.973,58.606,160.611
C02648=1013.995,64.129,-117.379,165.974,58.595,160.609
C02649=1013.999,64.379,-117.394,165.976,58.585,160.607
C02650=1014.004,64.628,-117.409,165.979,58.575,160.606
C02651=1014.009,64.878,-117.423,165.980,58.566,160.605
C02652=1014.013,65.127,-117.439,165.983,58.555,160.604
C02653=1014.018,65.377,-117.454,165.985,58.546,160.602
C02654=1014.022,65.627,-117.469,165.988,58.535,160.601
C02655=1014.027,65.876,-117.485,165.990,58.526,160.599
C02656=1014.032,66.125,-117.499,165.993,58.516,160.598
C02657=1014.036,66.375,-117.514,165.994,58.506,160.597
C02658=1014.041,66.624,-117.530,165.996,58.496,160.595
C02659=1014.045,66.874,-117.545,165.999,58.486,160.594
C02660=1014.050,67.124,-117.560,166.000,58.475,160.592
C02661=1014.055,67.373,-117.575,166.003,58.465,160.591
C02662=1014.059,67.623,-117.591,166.005,58.456,160.590
C02663=1014.064,67.872,-117.606,166.008,58.445,160.588
C02664=1014.068,68.122,-117.621,166.010,58.436,160.587
C02665=1014.073,68.371,-117.636,166.013,58.425,160.586
C02666=1014.077,68.620,-117.652,166.015,58.416,160.584
C02667=1014.082,68.869,-117.667,166.017,58.405,160.583
C02668=1014.086,69.119,-117.683,166.019,58.395,160.581
C02669=1014.091,69.369,-117.697,166.022,58.385,160.580
C02670=1014.096,69.618,-117.713,166.024,58.375,160.579
C02671=1014.100,69.868,-117.729,166.026,58.365,160.577
C02672=1014.105,70.117,-117.744,166.028,58.355,160.576
C02673=1014.109,70.367,-117.760,166.031,58.344,160.574
C02674=1014.114,70.616,-117.775,166.032,58.335,160.573
C02675=1014.118,70.866,-117.790,166.035,58.325,160.572
C02676=1014.123,71.116,-117.805,166.037,58.315,160.570
C02677=1014.128,71.365,-117.821,166.040,58.305,160.569
C02678=1014.133,71.614,-117.836,166.041,58.294,160.567
C02679=1014.137,71.864,-117.852,166.044,58.284,160.566
C02680=1014.141,72.114,-117.867,166.046,58.274,160.565
C02681=1014.146,72.363,-117.883,166.049,58.264,160.563
C02682=1014.151,72.612,-117.898,166.051,58.254,160.562
C02683=1014.156,72.862,-117.914,166.053,58.244,160.560
C02684=1014.159,73.111,-117.929,166.056,58.234,160.559
C02685=1014.163,73.361,-117.944,166.058,58.223,160.557
C02686=1014.168,73.610,-117.959,166.061,58.213,160.556
C02687=1014.173,73.860,-117.975,166.063,58.203,160.555
C02688=1014.178,74.139,-117.993,166.065,58.191,160.553
C02689=1014.183,74.420,-118.010,166.068,58.180,160.552
C02690=1014.188,74.700,-118.027,166.071,58.168,160.550
C02691=1014.195,74.980,-118.045,166.074,58.157,160.549
C02692=1014.199,75.229,-118.061,166.075,58.147,160.547
C02693=1014.203,75.479,-118.076,166.078,58.137,160.546
C02694=1014.208,75.728,-118.092,166.080,58.126,160.544
C02695=1014.213,75.978,-118.107,166.083,58.116,160.543
C02696=1014.217,76.227,-118.123,166.086,58.106,160.541
C02697=1014.222,76.477,-118.138,166.087,58.096,160.540
C02698=1014.226,76.726,-118.154,166.090,58.085,160.539
C02699=1014.231,76.976,-118.170,166.092,58.076,160.537
C02700=1014.235,77.225,-118.186,166.094,58.065,160.536
C02701=1014.239,77.475,-118.201,166.097,58.055,160.534
C02702=1014.243,77.724,-118.217,166.099,58.045,160.533
C02703=1014.249,77.974,-118.232,166.101,58.034,160.531
C02704=1014.253,78.223,-118.249,166.103,58.025,160.530
C02705=1014.257,78.472,-118.265,166.106,58.014,160.529
C02706=1014.262,78.722,-118.280,166.108,58.004,160.527
C02707=1014.266,78.971,-118.296,166.111,57.994,160.526
C02708=1014.270,79.221,-118.312,166.113,57.983,160.524
C02709=1014.275,79.470,-118.328,166.115,57.974,160.523
C02710=1014.279,79.719,-118.344,166.118,57.963,160.522
C02711=1014.284,79.969,-118.359,166.120,57.953,160.520
C02712=1014.289,80.218,-118.375,166.123,57.943,160.519
C02713=1014.293,80.468,-118.391,166.125,57.932,160.517
C02714=1014.298,80.718,-118.408,166.127,57.922,160.516
C02715=1014.302,80.967,-118.423,166.129,57.912,160.514
C02716=1014.307,81.217,-118.439,166.132,57.902,160.513
C02717=1014.311,81.466,-118.455,166.134,57.891,160.511
C02718=1014.316,81.715,-118.471,166.137,57.881,160.510
C02719=1014.321,81.965,-118.487,166.139,57.870,160.509
C02720=1014.325,82.214,-118.502,166.141,57.861,160.507
C02721=1014.329,82.464,-118.518,166.144,57.850,160.506
C02722=1014.334,82.713,-118.535,166.147,57.840,160.505
C02723=1014.338,82.962,-118.550,166.148,57.829,160.503
C02724=1014.343,83.212,-118.567,166.151,57.819,160.502
C02725=1014.348,83.461,-118.583,166.154,57.808,160.500
C02726=1014.352,83.711,-118.599,166.157,57.798,160.499
C02727=1014.356,83.961,-118.615,166.158,57.788,160.497
C02728=1014.362,84.209,-118.630,166.161,57.777,160.496
C02729=1014.366,84.459,-118.646,166.164,57.767,160.495
C02730=1014.370,84.708,-118.662,166.166,57.756,160.493
C02731=1014.375,84.959,-118.678,166.168,57.747,160.492
C02732=1014.380,85.208,-118.695,166.171,57.736,160.490
C02733=1014.384,85.457,-118.710,166.173,57.725,160.489
C02734=1014.388,85.707,-118.726,166.176,57.715,160.487
C02735=1014.393,85.956,-118.743,166.178,57.705,160.486
C02736=1014.398,86.205,-118.758,166.180,57.694,160.484
C02737=1014.402,86.455,-118.774,166.183,57.684,160.483
C02738=1014.408,86.704,-118.790,166.186,57.673,160.482
C02739=1014.412,86.954,-118.806,166.188,57.662,160.480
C02740=1014.417,87.203,-118.823,166.190,57.652,160.478
C02741=1014.421,87.452,-118.838,166.193,57.642,160.477
C02742=1014.425,87.702,-118.854,166.195,57.631,160.476
C02743=1014.430,87.952,-118.871,166.198,57.620,160.474
C02744=1014.435,88.201,-118.887,166.200,57.610,160.473
C02745=1014.440,88.450,-118.902,166.203,57.600,160.472
C02746=1014.444,88.699,-118.919,166.205,57.589,160.470
C02747=1014.448,88.949,-118.935,166.207,57.579,160.468
C02748=1014.453,89.199,-118.952,166.211,57.568,160.467
C02749=1014.458,89.448,-118.968,166.213,57.558,160.466
C02750=1014.462,89.697,-118.984,166.215,57.548,160.464
C02751=1014.467,89.946,-119.000,166.218,57.537,160.463
C02752=1014.472,90.227,-119.019,166.221,57.525,160.461
C02753=1014.477,90.507,-119.038,166.223,57.514,160.459
C02754=1014.481,90.788,-119.056,166.226,57.502,160.458
C02755=1014.487,91.068,-119.074,166.229,57.491,160.457
C02756=1014.491,91.318,-119.091,166.232,57.480,160.455
C02757=1014.496,91.567,-119.108,166.233,57.470,160.453
C02758=1014.500,91.816,-119.124,166.236,57.459,160.452
C02759=1014.505,92.065,-119.140,166.239,57.449,160.451
C02760=1014.509,92.316,-119.156,166.242,57.438,160.449
C02761=1014.513,92.565,-119.173,166.244,57.428,160.448
C02762=1014.518,92.814,-119.190,166.246,57.418,160.446
C02763=1014.522,93.063,-119.206,166.249,57.407,160.445
C02764=1014.527,93.313,-119.222,166.251,57.396,160.443
C02765=1014.531,93.562,-119.239,166.254,57.386,160.442
C02766=1014.536,93.812,-119.255,166.257,57.376,160.441
C02767=1014.540,94.061,-119.272,166.260,57.365,160.439
C02768=1014.545,94.311,-119.289,166.261,57.355,160.438
C02769=1014.550,94.560,-119.304,166.264,57.344,160.436
C02770=1014.554,94.809,-119.321,166.266,57.333,160.435
C02771=1014.558,95.058,-119.338,166.269,57.323,160.433
C02772=1014.563,95.308,-119.355,166.272,57.313,160.432
C02773=1014.568,95.558,-119.371,166.275,57.302,160.431
C02774=1014.572,95.806,-119.387,166.277,57.291,160.429
C02775=1014.577,96.056,-119.404,166.279,57.281,160.427
C02776=1014.581,96.306,-119.420,166.282,57.270,160.426
C02777=1014.586,96.555,-119.437,166.284,57.259,160.424
C02778=1014.591,96.805,-119.454,166.287,57.249,160.423
C02779=1014.596,97.054,-119.470,166.290,57.239,160.422
C02780=1014.599,97.304,-119.486,166.293,57.228,160.420
C02781=1014.604,97.553,-119.503,166.295,57.217,160.419
C02782=1014.609,97.802,-119.520,166.298,57.207,160.417
C02783=1014.614,98.051,-119.536,166.301,57.196,160.416
C02784=1014.618,98.302,-119.553,166.303,57.185,160.414
C02785=1014.622,98.551,-119.569,166.306,57.174,160.413
C02786=1014.627,98.800,-119.586,166.308,57.164,160.412
C02787=1014.632,99.049,-119.603,166.310,57.153,160.410
C02788=1014.636,99.299,-119.620,166.313,57.143,160.409
C02789=1014.640,99.548,-119.637,166.316,57.133,160.407
C02790=1014.645,99.797,-119.654,166.319,57.122,160.406
C02791=1014.649,100.047,-119.671,166.321,57.111,160.404
C02792=1014.654,100.296,-119.688,166.324,57.101,160.403
C02793=1014.658,100.546,-119.705,166.325,57.090,160.401
C02794=1014.663,100.795,-119.721,166.329,57.081,160.400
C02795=1014.667,101.045,-119.739,166.331,57.070,160.399
C02796=1014.672,101.294,-119.755,166.334,57.059,160.397
C02797=1014.676,101.543,-119.772,166.337,57.048,160.396
C02798=1014.681,101.792,-119.789,166.339,57.038,160.394
C02799=1014.685,102.042,-119.806,166.342,57.027,160.393
C02800=1014.690,102.291,-119.823,166.345,57.016,160.391
C02801=1014.694,102.541,-119.840,166.348,57.006,160.390
C02802=1014.699,102.790,-119.857,166.350,56.996,160.389
C02803=1014.703,103.040,-119.874,166.352,56.986,160.387
C02804=1014.708,103.289,-119.891,166.355,56.975,160.386
C02805=1014.712,103.539,-119.908,166.358,56.964,160.384
C02806=1014.717,103.787,-119.925,166.360,56.954,160.383
C02807=1014.721,104.037,-119.942,166.363,56.943,160.381
C02808=1014.726,104.286,-119.958,166.366,56.932,160.380
C02809=1014.730,104.536,-119.976,166.368,56.922,160.378
C02810=1014.735,104.785,-119.992,166.371,56.911,160.377
C02811=1014.739,105.035,-120.009,166.374,56.900,160.375
C02812=1014.744,105.284,-120.026,166.377,56.890,160.374
C02813=1014.748,105.534,-120.043,166.379,56.879,160.373
C02814=1014.753,105.782,-120.061,166.382,56.868,160.371
C02815=1014.757,106.032,-120.078,166.385,56.858,160.370
C02816=1014.763,106.313,-120.097,166.388,56.846,160.368
C02817=1014.767,106.593,-120.116,166.391,56.834,160.367
C02818=1014.772,106.874,-120.135,166.394,56.822,160.365
C02819=1014.777,107.154,-120.155,166.397,56.810,160.363
C02820=1014.782,107.403,-120.171,166.400,56.799,160.362
C02821=1014.787,107.653,-120.189,166.403,56.788,160.360
C02822=1014.791,107.902,-120.205,166.405,56.778,160.359
C02823=1014.796,108.152,-120.223,166.408,56.767,160.357
C02824=1014.800,108.401,-120.239,166.411,56.757,160.356
C02825=1014.805,108.650,-120.257,166.413,56.745,160.354
C02826=1014.810,108.899,-120.274,166.416,56.735,160.353
C02827=1014.814,109.149,-120.291,166.418,56.724,160.351
C02828=1014.818,109.398,-120.308,166.421,56.713,160.350
C02829=1014.823,109.648,-120.325,166.424,56.703,160.349
C02830=1014.827,109.897,-120.343,166.427,56.692,160.347
C02831=1014.832,110.147,-120.360,166.430,56.681,160.346
C02832=1014.836,110.396,-120.377,166.432,56.671,160.344
C02833=1014.841,110.645,-120.395,166.435,56.660,160.343
C02834=1014.846,110.895,-120.413,166.438,56.650,160.341
C02835=1014.850,111.144,-120.430,166.441,56.639,160.340
C02836=1014.855,111.393,-120.447,166.443,56.628,160.339
C02837=1014.859,111.643,-120.464,166.446,56.618,160.337
C02838=1014.863,111.893,-120.482,166.449,56.607,160.336
C02839=1014.868,112.141,-120.499,166.452,56.597,160.334
C02840=1014.872,112.391,-120.517,166.455,56.586,160.333
C02841=1014.876,112.640,-120.535,166.457,56.575,160.331
C02842=1014.881,112.890,-120.552,166.460,56.565,160.330
C02843=1014.885,113.138,-120.570,166.463,56.554,160.329
C02844=1014.889,113.388,-120.587,166.466,56.544,160.327
C02845=1014.894,113.638,-120.606,166.469,56.533,160.326
C02846=1014.898,113.887,-120.623,166.470,56.523,160.324
C02847=1014.903,114.136,-120.641,166.473,56.512,160.323
C02848=1014.907,114.386,-120.658,166.476,56.502,160.321
C02849=1014.912,114.635,-120.676,166.479,56.491,160.320
C02850=1014.915,114.884,-120.693,166.482,56.480,160.318
C02851=1014.920,115.134,-120.711,166.485,56.470,160.317
C02852=1014.925,115.383,-120.729,166.487,56.459,160.316
C02853=1014.929,115.632,-120.747,166.490,56.449,160.314
C02854=1014.934,115.882,-120.765,166.493,56.438,160.313
C02855=1014.937,116.131,-120.782,166.496,56.428,160.311
C02856=1014.942,116.380,-120.800,166.499,56.417,160.310
C02857=1014.947,116.630,-120.817,166.502,56.406,160.308
C02858=1014.951,116.879,-120.835,166.504,56.396,160.307
C02859=1014.956,117.128,-120.853,166.507,56.385,160.306
C02860=1014.960,117.377,-120.870,166.510,56.375,160.304
C02861=1014.964,117.627,-120.889,166.513,56.364,160.303
C02862=1014.969,117.876,-120.907,166.516,56.354,160.301
C02863=1014.973,118.125,-120.924,166.519,56.343,160.300
C02864=1014.978,118.375,-120.942,166.522,56.332,160.299
C02865=1014.982,118.625,-120.959,166.524,56.322,160.297
C02866=1014.986,118.873,-120.977,166.528,56.311,160.296
C02867=1014.991,119.123,-120.995,166.531,56.300,160.294
C02868=1014.996,119.373,-121.013,166.534,56.289,160.293
C02869=1015.000,119.621,-121.031,166.536,56.279,160.291
C02870=1015.005,119.871,-121.049,166.539,56.268,160.290
C02871=1015.009,120.121,-121.066,166.542,56.257,160.289
C02872=1015.013,120.369,-121.084,166.545,56.247,160.287
C02873=1015.018,120.619,-121.102,166.548,56.236,160.286
C02874=1015.023,120.869,-121.120,166.551,56.226,160.284
C02875=1015.027,121.117,-121.137,166.553,56.215,160.283
C02876=1015.032,121.367,-121.156,166.556,56.204,160.281
C02877=1015.036,121.616,-121.174,166.560,56.193,160.280
C02878=1015.040,121.865,-121.191,166.563,56.183,160.279
C02879=1015.045,122.115,-121.209,166.566,56.172,160.277
C02880=1015.050,122.395,-121.229,166.569,56.160,160.275
C02881=1015.055,122.676,-121.250,166.572,56.148,160.274
C02882=1015.060,122.956,-121.270,166.575,56.136,160.272
C02883=1015.065,123.237,-121.290,166.578,56.124,160.271
C02884=1015.069,123.487,-121.307,166.582,56.113,160.269
C02885=1015.074,123.736,-121.326,166.585,56.102,160.268
C02886=1015.079,123.985,-121.344,166.588,56.091,160.266
C02887=1015.083,124.235,-121.362,166.591,56.081,160.265
C02888=1015.087,124.484,-121.379,166.594,56.070,160.264
C02889=1015.092,124.733,-121.397,166.596,56.059,160.262
C02890=1015.097,124.983,-121.415,166.600,56.048,160.261
C02891=1015.102,125.232,-121.434,166.603,56.037,160.259
C02892=1015.106,125.481,-121.451,166.606,56.027,160.258
C02893=1015.110,125.731,-121.469,166.608,56.016,160.256
C02894=1015.115,125.980,-121.487,166.611,56.005,160.255
C02895=1015.120,126.229,-121.505,166.615,55.994,160.254
C02896=1015.124,126.478,-121.523,166.618,55.983,160.252
C02897=1015.129,126.727,-121.541,166.621,55.973,160.250
C02898=1015.133,126.977,-121.559,166.623,55.962,160.249
C02899=1015.138,127.227,-121.577,166.626,55.951,160.247
C02900=1015.143,127.476,-121.595,166.630,55.940,160.246
C02901=1015.147,127.725,-121.613,166.633,55.929,160.245
C02902=1015.152,127.974,-121.631,166.635,55.918,160.243
C02903=1015.156,128.223,-121.649,166.638,55.908,160.242
C02904=1015.161,128.473,-121.667,166.642,55.897,160.241
C02905=1015.166,128.722,-121.685,166.645,55.886,160.239
C02906=1015.171,128.972,-121.703,166.648,55.875,160.237
C02907=1015.175,129.221,-121.721,166.651,55.865,160.236
C02908=1015.179,129.470,-121.739,166.654,55.853,160.235
C02909=1015.184,129.720,-121.757,166.657,55.843,160.233
C02910=1015.188,129.969,-121.776,166.660,55.832,160.232
C02911=1015.192,130.219,-121.794,166.663,55.822,160.230
C02912=1015.197,130.467,-121.813,166.666,55.811,160.229
C02913=1015.202,130.717,-121.831,166.669,55.800,160.227
C02914=1015.206,130.966,-121.850,166.673,55.789,160.226
C02915=1015.210,131.215,-121.868,166.676,55.779,160.225
C02916=1015.214,131.465,-121.887,166.679,55.768,160.223
C02917=1015.219,131.714,-121.905,166.682,55.758,160.222
C02918=1015.224,131.963,-121.923,166.684,55.747,160.220
C02919=1015.228,132.213,-121.942,166.687,55.736,160.219
C02920=1015.233,132.462,-121.961,166.691,55.725,160.218
C02921=1015.237,132.710,-121.978,166.694,55.715,160.216
C02922=1015.241,132.960,-121.997,166.697,55.704,160.215
C02923=1015.246,133.209,-122.015,166.700,55.693,160.213
C02924=1015.250,133.459,-122.034,166.703,55.683,160.212
C02925=1015.255,133.708,-122.053,166.707,55.672,160.211
C02926=1015.260,133.957,-122.071,166.710,55.661,160.209
C02927=1015.264,134.207,-122.090,166.713,55.650,160.208
C02928=1015.269,134.456,-122.108,166.716,55.640,160.206
C02929=1015.273,134.706,-122.127,166.720,55.629,160.205
C02930=1015.277,134.954,-122.145,166.722,55.618,160.203
C02931=1015.282,135.203,-122.163,166.725,55.607,160.202
C02932=1015.286,135.453,-122.182,166.728,55.597,160.201
C02933=1015.291,135.702,-122.200,166.731,55.587,160.199
C02934=1015.295,135.951,-122.220,166.735,55.575,160.198
C02935=1015.300,136.201,-122.238,166.738,55.565,160.197
C02936=1015.304,136.450,-122.257,166.741,55.554,160.195
C02937=1015.309,136.699,-122.276,166.744,55.544,160.194
C02938=1015.313,136.949,-122.294,166.748,55.532,160.192
C02939=1015.318,137.198,-122.313,166.751,55.522,160.191
C02940=1015.322,137.447,-122.332,166.754,55.511,160.190
C02941=1015.327,137.696,-122.350,166.756,55.500,160.188
C02942=1015.331,137.946,-122.369,166.761,55.489,160.187
C02943=1015.336,138.195,-122.388,166.764,55.479,160.185
C02944=1015.341,138.476,-122.409,166.767,55.467,160.184
C02945=1015.346,138.757,-122.431,166.770,55.455,160.182
C02946=1015.351,139.036,-122.452,166.774,55.444,160.181
C02947=1015.356,139.318,-122.473,166.778,55.431,160.179
C02948=1015.361,139.567,-122.492,166.781,55.421,160.178
C02949=1015.365,139.816,-122.511,166.784,55.410,160.176
C02950=1015.369,140.065,-122.530,166.787,55.399,160.175
C02951=1015.374,140.315,-122.548,166.791,55.388,160.173
C02952=1015.378,140.564,-122.568,166.794,55.378,160.172
C02953=1015.382,140.813,-122.586,166.797,55.367,160.171
C02954=1015.387,141.062,-122.605,166.800,55.356,160.169
C02955=1015.391,141.312,-122.624,166.804,55.346,160.168
C02956=1015.396,141.561,-122.643,166.807,55.335,160.167
C02957=1015.400,141.810,-122.662,166.810,55.325,160.165
C02958=1015.405,142.059,-122.681,166.813,55.314,160.164
C02959=1015.409,142.308,-122.701,166.817,55.303,160.162
C02960=1015.414,142.558,-122.719,166.820,55.293,160.161
C02961=1015.418,142.807,-122.738,166.823,55.282,160.160
C02962=1015.422,143.056,-122.757,166.827,55.271,160.158
C02963=1015.427,143.305,-122.776,166.830,55.260,160.157
C02964=1015.431,143.555,-122.795,166.833,55.250,160.155
C02965=1015.436,143.804,-122.814,166.837,55.238,160.154
C02966=1015.441,144.052,-122.833,166.840,55.228,160.153
C02967=1015.445,144.302,-122.852,166.843,55.218,160.151
C02968=1015.449,144.551,-122.871,166.846,55.207,160.150
C02969=1015.455,144.801,-122.890,166.850,55.196,160.148
C02970=1015.459,145.050,-122.909,166.853,55.185,160.147
C02971=1015.463,145.299,-122.929,166.856,55.174,160.145
C02972=1015.468,145.570,-122.949,166.860,55.163,160.144
C02973=1015.473,145.840,-122.970,166.863,55.151,160.143
C02974=1015.478,146.110,-122.991,166.867,55.140,160.141
C02975=1015.482,146.382,-123.011,166.871,55.129,160.140
C02976=1015.487,146.631,-123.031,166.875,55.118,160.138
C02977=1015.492,146.879,-123.050,166.878,55.107,160.137
C02978=1015.497,147.129,-123.070,166.881,55.096,160.135
C02979=1015.501,147.379,-123.088,166.885,55.086,160.134
C02980=1015.505,147.628,-123.108,166.888,55.075,160.133
C02981=1015.509,147.877,-123.127,166.891,55.064,160.131
C02982=1015.514,148.126,-123.147,166.895,55.054,160.130
C02983=1015.518,148.375,-123.166,166.898,55.043,160.129
C02984=1015.522,148.624,-123.186,166.902,55.033,160.127
C02985=1015.527,148.874,-123.205,166.905,55.023,160.126
C02986=1015.531,149.123,-123.224,166.908,55.011,160.125
C02987=1015.536,149.372,-123.244,166.912,55.001,160.123
C02988=1015.541,149.621,-123.263,166.915,54.990,160.122
C02989=1015.545,149.870,-123.282,166.919,54.980,160.121
C02990=1015.550,150.119,-123.302,166.922,54.969,160.119
C02991=1015.555,150.369,-123.322,166.925,54.958,160.118
C02992=1015.559,150.618,-123.341,166.929,54.948,160.117
C02993=1015.563,150.867,-123.360,166.932,54.937,160.115
C02994=1015.568,151.116,-123.380,166.935,54.926,160.114
C02995=1015.572,151.365,-123.399,166.940,54.916,160.112
C02996=1015.577,151.615,-123.419,166.943,54.905,160.111
C02997=1015.581,151.865,-123.438,166.945,54.894,160.109
C02998=1015.585,152.114,-123.457,166.950,54.884,160.108
C02999=1015.590,152.363,-123.477,166.953,54.873,160.107
C03000=1015.594,152.612,-123.496,166.957,54.863,160.106
C03001=1015.599,152.861,-123.516,166.960,54.852,160.104
C03002=1015.603,153.110,-123.536,166.963,54.841,160.103
C03003=1015.608,153.359,-123.556,166.966,54.831,160.101
C03004=1015.612,153.608,-123.575,166.971,54.820,160.100
C03005=1015.617,153.858,-123.595,166.974,54.809,160.099
C03006=1015.622,154.107,-123.615,166.978,54.799,160.097
C03007=1015.625,154.356,-123.635,166.981,54.788,160.096
C03008=1015.630,154.615,-123.655,166.985,54.777,160.095
C03009=1015.635,154.875,-123.676,166.988,54.767,160.093
C03010=1015.640,155.134,-123.696,166.992,54.755,160.092
C03011=1015.644,155.392,-123.717,166.996,54.744,160.090
C03012=1015.649,155.642,-123.736,166.999,54.733,160.089
C03013=1015.653,155.891,-123.756,167.002,54.723,160.088
C03014=1015.658,156.140,-123.775,167.007,54.713,160.087
C03015=1015.662,156.389,-123.795,167.009,54.702,160.085
C03016=1015.667,156.639,-123.815,167.014,54.691,160.084
C03017=1015.671,156.888,-123.835,167.017,54.681,160.082
C03018=1015.675,157.137,-123.855,167.020,54.670,160.081
C03019=1015.680,157.387,-123.875,167.024,54.659,160.080
C03020=1015.685,157.636,-123.894,167.027,54.649,160.078
C03021=1015.689,157.885,-123.914,167.032,54.638,160.077
C03022=1015.694,158.134,-123.934,167.035,54.627,160.076
C03023=1015.698,158.383,-123.954,167.039,54.616,160.074
C03024=1015.702,158.632,-123.974,167.042,54.606,160.073
C03025=1015.707,158.881,-123.994,167.046,54.596,160.072
C03026=1015.711,159.131,-124.014,167.049,54.586,160.070
C03027=1015.715,159.380,-124.036,167.053,54.575,160.069
C03028=1015.720,159.629,-124.055,167.057,54.565,160.068
C03029=1015.724,159.878,-124.076,167.060,54.555,160.067
C03030=1015.729,160.128,-124.096,167.063,54.544,160.065
C03031=1015.733,160.376,-124.116,167.068,54.534,160.064
C03032=1015.736,160.626,-124.137,167.071,54.523,160.063
C03033=1015.741,160.875,-124.157,167.074,54.513,160.061
C03034=1015.745,161.124,-124.177,167.079,54.503,160.060
C03035=1015.750,161.373,-124.197,167.081,54.492,160.059
C03036=1015.754,161.623,-124.218,167.085,54.481,160.057
C03037=1015.759,161.871,-124.238,167.089,54.471,160.056
C03038=1015.762,162.120,-124.258,167.092,54.461,160.055
C03039=1015.767,162.370,-124.279,167.096,54.450,160.053
C03040=1015.771,162.618,-124.299,167.100,54.440,160.052
C03041=1015.776,162.868,-124.320,167.104,54.429,160.051
C03042=1015.780,163.117,-124.340,167.107,54.419,160.050
C03043=1015.784,163.366,-124.360,167.111,54.409,160.048
C03044=1015.788,163.616,-124.381,167.115,54.398,160.047
C03045=1015.793,163.864,-124.401,167.118,54.388,160.046
C03046=1015.797,164.114,-124.422,167.122,54.378,160.045
C03047=1015.802,164.363,-124.442,167.125,54.367,160.043
C03048=1015.806,164.611,-124.463,167.129,54.356,160.042
C03049=1015.811,164.861,-124.483,167.133,54.346,160.041
C03050=1015.815,165.110,-124.503,167.136,54.336,160.039
C03051=1015.819,165.359,-124.525,167.141,54.325,160.038
C03052=1015.824,165.608,-124.544,167.144,54.315,160.037
C03053=1015.828,165.858,-124.565,167.148,54.305,160.035
C03054=1015.833,166.106,-124.585,167.152,54.294,160.034
C03055=1015.837,166.356,-124.606,167.155,54.284,160.033
C03056=1015.841,166.605,-124.627,167.159,54.273,160.031
C03057=1015.846,166.854,-124.647,167.163,54.262,160.030
C03058=1015.850,167.103,-124.667,167.167,54.252,160.029
C03059=1015.855,167.352,-124.688,167.170,54.242,160.028
C03060=1015.859,167.601,-124.709,167.174,54.231,160.026
C03061=1015.864,167.850,-124.729,167.178,54.221,160.025
C03062=1015.868,168.100,-124.749,167.182,54.211,160.024
C03063=1015.872,168.349,-124.770,167.186,54.199,160.022
C03064=1015.877,168.598,-124.790,167.189,54.189,160.021
C03065=1015.881,168.847,-124.812,167.194,54.179,160.020
C03066=1015.886,169.095,-124.832,167.197,54.169,160.019
C03067=1015.890,169.345,-124.852,167.201,54.158,160.017
C03068=1015.894,169.594,-124.873,167.205,54.148,160.016
C03069=1015.899,169.843,-124.894,167.209,54.137,160.015
C03070=1015.903,170.092,-124.914,167.212,54.126,160.013
C03071=1015.909,170.341,-124.935,167.217,54.116,160.012
C03072=1015.913,170.622,-124.958,167.221,54.105,160.011
C03073=1015.918,170.902,-124.981,167.225,54.092,160.009
C03074=1015.924,171.182,-125.005,167.229,54.081,160.008
C03075=1015.928,171.462,-125.028,167.234,54.069,160.006
C03076=1015.933,171.712,-125.049,167.237,54.058,160.005
C03077=1015.937,171.960,-125.069,167.242,54.048,160.004
C03078=1015.943,172.209,-125.090,167.245,54.038,160.002
C03079=1015.947,172.459,-125.111,167.250,54.027,160.001
C03080=1015.951,172.708,-125.131,167.254,54.017,160.000
C03081=1015.956,172.957,-125.152,167.257,54.006,159.998
C03082=1015.960,173.206,-125.172,167.261,53.995,159.997
C03083=1015.965,173.455,-125.193,167.265,53.985,159.996
C03084=1015.970,173.705,-125.214,167.269,53.975,159.995
C03085=1015.974,173.953,-125.235,167.273,53.965,159.994
C03086=1015.979,174.203,-125.256,167.277,53.953,159.992
C03087=1015.983,174.452,-125.277,167.281,53.943,159.991
C03088=1015.988,174.700,-125.297,167.285,53.933,159.990
C03089=1015.993,174.950,-125.318,167.289,53.922,159.988
C03090=1015.997,175.199,-125.339,167.293,53.912,159.987
C03091=1016.002,175.448,-125.359,167.297,53.901,159.986
C03092=1016.006,175.697,-125.380,167.300,53.891,159.984
C03093=1016.011,175.946,-125.401,167.305,53.880,159.983
C03094=1016.015,176.195,-125.422,167.309,53.870,159.982
C03095=1016.020,176.444,-125.443,167.313,53.860,159.981
C03096=1016.025,176.694,-125.464,167.317,53.848,159.979
C03097=1016.030,176.943,-125.485,167.321,53.838,159.978
C03098=1016.034,177.192,-125.505,167.325,53.828,159.977
C03099=1016.039,177.441,-125.526,167.329,53.817,159.976
C03100=1016.043,177.690,-125.547,167.334,53.807,159.974
C03101=1016.049,177.939,-125.568,167.337,53.796,159.973
C03102=1016.053,178.188,-125.589,167.342,53.786,159.972
C03103=1016.057,178.437,-125.610,167.345,53.775,159.970
C03104=1016.063,178.686,-125.631,167.350,53.765,159.969
C03105=1016.067,178.936,-125.652,167.354,53.754,159.968
C03106=1016.072,179.184,-125.672,167.357,53.744,159.967
C03107=1016.076,179.433,-125.693,167.362,53.733,159.965
C03108=1016.081,179.683,-125.715,167.366,53.723,159.964
C03109=1016.086,179.931,-125.736,167.371,53.712,159.963
C03110=1016.091,180.181,-125.757,167.374,53.701,159.961
C03111=1016.096,180.429,-125.777,167.378,53.691,159.960
C03112=1016.100,180.679,-125.798,167.383,53.681,159.959
C03113=1016.105,180.928,-125.819,167.387,53.670,159.958
C03114=1016.110,181.177,-125.841,167.391,53.659,159.956
C03115=1016.115,181.426,-125.862,167.395,53.649,159.955
C03116=1016.119,181.675,-125.883,167.400,53.638,159.954
C03117=1016.123,181.924,-125.904,167.403,53.628,159.953
C03118=1016.128,182.173,-125.926,167.408,53.618,159.952
C03119=1016.132,182.422,-125.947,167.411,53.608,159.950
C03120=1016.137,182.672,-125.969,167.416,53.597,159.949
C03121=1016.141,182.921,-125.990,167.420,53.587,159.948
C03122=1016.146,183.170,-126.012,167.425,53.578,159.947
C03123=1016.150,183.419,-126.035,167.428,53.568,159.946
C03124=1016.154,183.668,-126.056,167.433,53.557,159.944
C03125=1016.159,183.916,-126.077,167.436,53.547,159.943
C03126=1016.164,184.165,-126.099,167.441,53.537,159.942
C03127=1016.167,184.415,-126.121,167.444,53.527,159.941
C03128=1016.172,184.664,-126.143,167.449,53.516,159.939
C03129=1016.177,184.913,-126.164,167.453,53.506,159.938
C03130=1016.181,185.161,-126.186,167.457,53.496,159.937
C03131=1016.185,185.410,-126.208,167.462,53.485,159.936
C03132=1016.189,185.660,-126.229,167.465,53.475,159.934
C03133=1016.194,185.909,-126.251,167.471,53.465,159.934
C03134=1016.199,186.158,-126.273,167.474,53.455,159.932
C03135=1016.203,186.407,-126.295,167.479,53.445,159.931
C03136=1016.208,186.687,-126.319,167.484,53.434,159.930
C03137=1016.214,186.967,-126.344,167.488,53.422,159.928
C03138=1016.218,187.247,-126.369,167.493,53.410,159.927
C03139=1016.223,187.527,-126.393,167.498,53.399,159.926
C03140=1016.228,187.776,-126.415,167.502,53.389,159.924
C03141=1016.233,188.025,-126.437,167.506,53.378,159.923
C03142=1016.237,188.274,-126.458,167.511,53.368,159.922
C03143=1016.241,188.523,-126.480,167.514,53.358,159.921
C03144=1016.246,188.772,-126.502,167.520,53.348,159.920
C03145=1016.250,189.021,-126.525,167.524,53.338,159.919
C03146=1016.255,189.270,-126.546,167.528,53.328,159.917
C03147=1016.260,189.519,-126.568,167.532,53.317,159.916
C03148=1016.264,189.768,-126.589,167.537,53.307,159.915
C03149=1016.269,190.017,-126.612,167.541,53.297,159.914
C03150=1016.273,190.266,-126.634,167.545,53.287,159.912
C03151=1016.278,190.515,-126.656,167.550,53.276,159.911
C03152=1016.283,190.764,-126.677,167.554,53.266,159.910
C03153=1016.287,191.013,-126.700,167.558,53.256,159.909
C03154=1016.292,191.262,-126.721,167.563,53.246,159.908
C03155=1016.296,191.511,-126.743,167.567,53.236,159.906
C03156=1016.301,191.760,-126.765,167.572,53.226,159.905
C03157=1016.305,192.009,-126.787,167.576,53.216,159.904
C03158=1016.310,192.258,-126.809,167.581,53.205,159.903
C03159=1016.315,192.507,-126.831,167.585,53.195,159.902
C03160=1016.319,192.756,-126.853,167.589,53.185,159.901
C03161=1016.324,193.005,-126.875,167.594,53.175,159.899
C03162=1016.329,193.254,-126.898,167.598,53.165,159.898
C03163=1016.333,193.503,-126.920,167.602,53.154,159.897
C03164=1016.338,193.752,-126.942,167.607,53.144,159.896
C03165=1016.343,194.001,-126.964,167.612,53.134,159.895
C03166=1016.348,194.250,-126.986,167.615,53.124,159.893
C03167=1016.352,194.499,-127.008,167.620,53.113,159.892
C03168=1016.357,194.748,-127.030,167.625,53.103,159.891
C03169=1016.362,194.996,-127.052,167.630,53.093,159.890
C03170=1016.366,195.246,-127.074,167.635,53.083,159.889
C03171=1016.371,195.495,-127.096,167.638,53.073,159.888
C03172=1016.376,195.744,-127.118,167.643,53.063,159.886
C03173=1016.380,195.993,-127.141,167.648,53.052,159.885
C03174=1016.385,196.242,-127.163,167.652,53.042,159.884
C03175=1016.390,196.490,-127.185,167.657,53.032,159.883
C03176=1016.395,196.739,-127.207,167.661,53.022,159.882
C03177=1016.399,196.989,-127.230,167.665,53.011,159.880
C03178=1016.404,197.237,-127.252,167.670,53.001,159.879
C03179=1016.409,197.486,-127.274,167.675,52.991,159.878
C03180=1016.413,197.735,-127.296,167.680,52.980,159.877
C03181=1016.419,197.985,-127.318,167.685,52.971,159.876
C03182=1016.424,198.233,-127.341,167.688,52.961,159.875
C03183=1016.428,198.482,-127.363,167.693,52.951,159.874
C03184=1016.433,198.731,-127.385,167.698,52.940,159.872
C03185=1016.438,198.980,-127.407,167.703,52.930,159.871
C03186=1016.442,199.230,-127.430,167.707,52.920,159.870
C03187=1016.447,199.478,-127.452,167.712,52.909,159.869
C03188=1016.451,199.727,-127.475,167.716,52.900,159.868
C03189=1016.456,199.975,-127.498,167.721,52.890,159.867
C03190=1016.461,200.225,-127.520,167.726,52.880,159.866
C03191=1016.465,200.474,-127.543,167.730,52.869,159.864
C03192=1016.470,200.723,-127.566,167.735,52.860,159.863
C03193=1016.475,200.972,-127.588,167.739,52.850,159.862
C03194=1016.480,201.221,-127.611,167.744,52.840,159.861
C03195=1016.484,201.470,-127.634,167.749,52.830,159.860
C03196=1016.489,201.718,-127.656,167.754,52.820,159.859
C03197=1016.493,201.968,-127.679,167.758,52.810,159.858
C03198=1016.498,202.216,-127.702,167.763,52.799,159.856
C03199=1016.503,202.465,-127.724,167.768,52.790,159.855
C03200=1016.527,203.705,-127.840,168.266,52.861,159.972
C03201=1016.532,203.944,-127.864,168.271,52.852,159.971
C03202=1016.538,204.183,-127.887,168.274,52.843,159.969
C03203=1016.544,204.421,-127.910,168.279,52.835,159.969
C03204=1016.549,204.659,-127.933,168.282,52.827,159.968
C03205=1016.555,204.898,-127.957,168.287,52.818,159.967
C03206=1016.560,205.136,-127.979,168.290,52.810,159.966
C03207=1016.565,205.375,-128.004,168.294,52.801,159.964
C03208=1016.571,205.625,-128.028,168.298,52.793,159.963
C03209=1016.576,205.872,-128.053,168.302,52.784,159.962
C03210=1016.582,206.121,-128.078,168.307,52.775,159.961
C03211=1016.588,206.370,-128.102,168.311,52.767,159.960
C03212=1016.593,206.619,-128.126,168.314,52.758,159.959
C03213=1016.599,206.868,-128.152,168.319,52.749,159.958
C03214=1016.604,207.116,-128.176,168.323,52.740,159.957
C03215=1016.611,207.365,-128.200,168.327,52.732,159.956
C03216=1016.616,207.613,-128.226,168.331,52.724,159.955
C03217=1016.621,207.862,-128.250,168.335,52.715,159.954
C03218=1016.627,208.111,-128.274,168.340,52.706,159.953
C03219=1016.633,208.359,-128.299,168.343,52.698,159.952
C03220=1016.639,208.609,-128.324,168.347,52.689,159.951
C03221=1016.644,208.857,-128.349,168.352,52.680,159.950
C03222=1016.650,209.106,-128.374,168.356,52.672,159.949
C03223=1016.655,209.354,-128.398,168.360,52.663,159.948
C03224=1016.662,209.603,-128.423,168.364,52.655,159.947
C03225=1016.667,209.852,-128.447,168.368,52.647,159.946
C03226=1016.673,210.100,-128.473,168.372,52.638,159.945
C03227=1016.678,210.349,-128.498,168.377,52.630,159.944
C03228=1016.684,210.598,-128.523,168.380,52.621,159.943
C03229=1016.689,210.847,-128.547,168.385,52.613,159.942
C03230=1016.695,211.095,-128.573,168.388,52.605,159.941
C03231=1016.701,211.344,-128.599,168.393,52.596,159.940
C03232=1016.706,211.593,-128.623,168.397,52.588,159.939
C03233=1016.712,211.841,-128.648,168.401,52.580,159.938
C03234=1016.718,212.090,-128.672,168.406,52.571,159.937
C03235=1016.723,212.339,-128.698,168.409,52.563,159.936
C03236=1016.728,212.588,-128.723,168.414,52.555,159.935
C03237=1016.735,212.836,-128.748,168.417,52.547,159.934
C03238=1016.740,213.084,-128.773,168.422,52.538,159.933
C03239=1016.745,213.334,-128.798,168.427,52.530,159.933
C03240=1016.752,213.582,-128.823,168.430,52.522,159.931
C03241=1016.757,213.830,-128.848,168.435,52.513,159.931
C03242=1016.763,214.080,-128.873,168.438,52.505,159.930
C03243=1016.769,214.329,-128.899,168.443,52.497,159.929
C03244=1016.774,214.577,-128.924,168.447,52.489,159.928
C03245=1016.780,214.826,-128.949,168.451,52.480,159.927
C03246=1016.786,215.074,-128.974,168.455,52.472,159.926
C03247=1016.791,215.323,-128.999,168.459,52.464,159.925
C03248=1016.797,215.572,-129.025,168.463,52.456,159.924
C03249=1016.803,215.820,-129.049,168.468,52.447,159.923
C03250=1016.808,216.069,-129.075,168.471,52.439,159.922
C03251=1016.814,216.318,-129.100,168.476,52.431,159.921
C03252=1016.820,216.566,-129.125,168.481,52.423,159.920
C03253=1016.826,216.815,-129.150,168.484,52.415,159.919
C03254=1016.831,217.064,-129.176,168.489,52.407,159.918
C03255=1016.838,217.313,-129.201,168.493,52.399,159.917
C03256=1016.843,217.561,-129.226,168.497,52.390,159.916
C03257=1016.849,217.809,-129.252,168.501,52.382,159.915
C03258=1016.854,218.058,-129.277,168.506,52.375,159.915
C03259=1016.860,218.306,-129.302,168.510,52.367,159.914
C03260=1016.866,218.544,-129.326,168.514,52.359,159.913
C03261=1016.871,218.781,-129.351,168.517,52.351,159.912
C03262=1016.876,219.017,-129.375,168.521,52.344,159.911
C03263=1016.882,219.254,-129.399,168.525,52.336,159.910
C03264=1016.887,219.491,-129.424,168.529,52.329,159.909
C03265=1016.892,219.728,-129.448,168.533,52.321,159.908
C03266=1016.898,219.964,-129.473,168.537,52.314,159.908
C03267=1016.903,220.202,-129.497,168.541,52.306,159.907
C03268=1016.909,220.451,-129.523,168.546,52.298,159.906
C03269=1016.914,220.699,-129.548,168.550,52.291,159.905
C03270=1016.920,220.947,-129.573,168.554,52.283,159.904
C03271=1016.926,221.196,-129.600,168.559,52.275,159.903
C03272=1016.932,221.444,-129.625,168.562,52.267,159.902
C03273=1016.938,221.693,-129.651,168.567,52.259,159.902
C03274=1016.943,221.941,-129.676,168.571,52.251,159.901
C03275=1016.949,222.190,-129.702,168.575,52.244,159.900
C03276=1016.954,222.439,-129.728,168.580,52.236,159.899
C03277=1016.960,222.688,-129.754,168.584,52.228,159.898
C03278=1016.966,222.937,-129.779,168.587,52.220,159.897
C03279=1016.972,223.184,-129.805,168.592,52.213,159.896
C03280=1016.977,223.433,-129.831,168.596,52.205,159.895
C03281=1016.983,223.682,-129.856,168.600,52.197,159.895
C03282=1016.989,223.931,-129.882,168.605,52.190,159.894
C03283=1016.994,224.180,-129.908,168.609,52.182,159.893
C03284=1017.001,224.429,-129.934,168.614,52.174,159.892
C03285=1017.006,224.677,-129.960,168.618,52.166,159.891
C03286=1017.012,224.925,-129.985,168.622,52.159,159.890
C03287=1017.017,225.174,-130.011,168.627,52.151,159.890
C03288=1017.024,225.423,-130.037,168.631,52.143,159.889
C03289=1017.029,225.671,-130.063,168.635,52.136,159.888
C03290=1017.035,225.920,-130.089,168.640,52.128,159.887
C03291=1017.041,226.169,-130.114,168.643,52.120,159.886
C03292=1017.047,226.417,-130.141,168.647,52.113,159.885
C03293=1017.052,226.666,-130.167,168.652,52.105,159.885
C03294=1017.058,226.915,-130.192,168.657,52.098,159.884
C03295=1017.064,227.162,-130.219,168.661,52.090,159.883
C03296=1017.069,227.411,-130.245,168.664,52.082,159.882
C03297=1017.075,227.660,-130.271,168.669,52.075,159.881
C03298=1017.080,227.909,-130.297,168.674,52.067,159.881
C03299=1017.087,228.157,-130.323,168.678,52.060,159.880
C03300=1017.092,228.406,-130.349,168.682,52.053,159.879
C03301=1017.098,228.654,-130.376,168.686,52.046,159.878
C03302=1017.104,228.903,-130.402,168.691,52.038,159.878
C03303=1017.109,229.151,-130.428,168.695,52.031,159.877
C03304=1017.115,229.400,-130.454,168.699,52.023,159.876
C03305=1017.121,229.648,-130.480,168.703,52.016,159.875
C03306=1017.127,229.897,-130.507,168.707,52.009,159.874
C03307=1017.133,230.146,-130.533,168.713,52.001,159.874
C03308=1017.138,230.394,-130.560,168.717,51.994,159.873
C03309=1017.144,230.643,-130.586,168.721,51.987,159.872
C03310=1017.150,230.891,-130.612,168.725,51.979,159.871
C03311=1017.155,231.140,-130.639,168.729,51.972,159.870
C03312=1017.161,231.389,-130.665,168.733,51.965,159.870
C03313=1017.167,231.637,-130.691,168.738,51.957,159.869
C03314=1017.172,231.885,-130.718,168.742,51.950,159.868
C03315=1017.178,232.134,-130.745,168.746,51.943,159.867
C03316=1017.184,232.383,-130.771,168.751,51.936,159.867
C03317=1017.189,232.631,-130.797,168.755,51.929,159.866
C03318=1017.195,232.880,-130.824,168.759,51.921,159.865
C03319=1017.201,233.128,-130.851,168.763,51.914,159.864
C03320=1017.206,233.361,-130.875,168.768,51.908,159.864
C03321=1017.212,233.594,-130.899,168.772,51.900,159.863
C03322=1017.217,233.826,-130.925,168.777,51.894,159.862
C03323=1017.222,234.059,-130.949,168.780,51.887,159.862
C03324=1017.228,234.291,-130.975,168.784,51.880,159.861
C03325=1017.234,234.524,-130.999,168.789,51.874,159.860
C03326=1017.238,234.758,-131.024,168.792,51.867,159.860
C03327=1017.244,234.990,-131.049,168.796,51.860,159.859
C03328=1017.250,235.238,-131.076,168.801,51.853,159.858
C03329=1017.256,235.487,-131.102,168.805,51.846,159.858
C03330=1017.261,235.736,-131.128,168.809,51.839,159.857
C03331=1017.267,235.984,-131.155,168.813,51.832,159.856
C03332=1017.273,236.232,-131.182,168.819,51.825,159.855
C03333=1017.279,236.481,-131.209,168.823,51.818,159.855
C03334=1017.285,236.730,-131.235,168.827,51.810,159.854
C03335=1017.291,236.978,-131.262,168.832,51.804,159.853
C03336=1017.296,237.226,-131.289,168.836,51.797,159.852
C03337=1017.302,237.475,-131.315,168.841,51.790,159.852
C03338=1017.308,237.723,-131.342,168.845,51.783,159.851
C03339=1017.314,237.972,-131.369,168.849,51.776,159.850
C03340=1017.320,238.221,-131.396,168.853,51.769,159.850
C03341=1017.326,238.469,-131.422,168.858,51.762,159.849
C03342=1017.332,238.717,-131.449,168.862,51.755,159.848
C03343=1017.338,238.966,-131.476,168.867,51.748,159.848
C03344=1017.343,239.214,-131.503,168.872,51.741,159.847
C03345=1017.349,239.463,-131.530,168.876,51.734,159.846
C03346=1017.355,239.711,-131.557,168.881,51.727,159.846
C03347=1017.360,239.960,-131.584,168.885,51.721,159.845
C03348=1017.366,240.208,-131.611,168.889,51.713,159.844
C03349=1017.372,240.456,-131.638,168.894,51.707,159.844
C03350=1017.378,240.705,-131.666,168.898,51.700,159.843
C03351=1017.383,240.954,-131.693,168.903,51.693,159.842
C03352=1017.389,241.202,-131.719,168.907,51.687,159.842
C03353=1017.394,241.450,-131.747,168.912,51.680,159.841
C03354=1017.401,241.699,-131.774,168.916,51.673,159.840
C03355=1017.407,241.947,-131.801,168.920,51.666,159.840
C03356=1017.412,242.196,-131.828,168.925,51.660,159.839
C03357=1017.418,242.444,-131.856,168.928,51.653,159.838
C03358=1017.424,242.693,-131.883,168.933,51.646,159.838
C03359=1017.429,242.942,-131.910,168.937,51.640,159.837
C03360=1017.435,243.189,-131.937,168.942,51.633,159.837
C03361=1017.441,243.439,-131.965,168.946,51.627,159.836
C03362=1017.447,243.686,-131.992,168.951,51.619,159.835
C03363=1017.452,243.935,-132.019,168.955,51.613,159.835
C03364=1017.457,244.183,-132.047,168.960,51.606,159.834
C03365=1017.464,244.432,-132.074,168.964,51.600,159.833
C03366=1017.469,244.680,-132.102,168.969,51.593,159.833
C03367=1017.475,244.928,-132.130,168.974,51.587,159.832
C03368=1017.481,245.177,-132.157,168.978,51.580,159.832
C03369=1017.486,245.425,-132.185,168.983,51.574,159.831
C03370=1017.492,245.674,-132.212,168.986,51.567,159.830
C03371=1017.498,245.923,-132.240,168.991,51.561,159.830
C03372=1017.504,246.171,-132.267,168.995,51.554,159.829
C03373=1017.509,246.419,-132.295,169.000,51.548,159.829
C03374=1017.515,246.668,-132.323,169.005,51.541,159.828
C03375=1017.521,246.916,-132.350,169.009,51.535,159.827
C03376=1017.527,247.165,-132.378,169.014,51.528,159.827
C03377=1017.532,247.413,-132.406,169.018,51.522,159.826
C03378=1017.538,247.661,-132.433,169.023,51.515,159.826
C03379=1017.544,247.910,-132.461,169.027,51.509,159.825
C03380=1017.550,248.139,-132.486,169.032,51.503,159.825
C03381=1017.554,248.368,-132.512,169.036,51.498,159.824
C03382=1017.559,248.598,-132.538,169.040,51.491,159.824
C03383=1017.565,248.827,-132.563,169.044,51.486,159.823
C03384=1017.571,249.057,-132.589,169.048,51.480,159.822
C03385=1017.576,249.286,-132.614,169.053,51.474,159.822
C03386=1017.582,249.516,-132.640,169.056,51.468,159.821
C03387=1017.586,249.744,-132.665,169.060,51.462,159.821
C03388=1017.592,249.993,-132.693,169.065,51.456,159.820
C03389=1017.598,250.241,-132.721,169.070,51.449,159.820
C03390=1017.604,250.490,-132.749,169.075,51.443,159.819
C03391=1017.610,250.738,-132.777,169.079,51.437,159.819
C03392=1017.616,250.987,-132.804,169.084,51.430,159.818
C03393=1017.621,251.235,-132.832,169.088,51.424,159.818
C03394=1017.627,251.484,-132.860,169.092,51.418,159.817
C03395=1017.633,251.731,-132.888,169.097,51.412,159.816
C03396=1017.639,251.980,-132.916,169.102,51.405,159.816
C03397=1017.646,252.228,-132.944,169.106,51.399,159.815
C03398=1017.651,252.477,-132.972,169.111,51.393,159.815
C03399=1017.657,252.726,-132.999,169.116,51.386,159.814
C03400=1017.663,252.974,-133.027,169.120,51.380,159.814
C03401=1017.669,253.222,-133.055,169.125,51.374,159.813
C03402=1017.674,253.470,-133.083,169.129,51.368,159.813
C03403=1017.681,253.719,-133.111,169.134,51.361,159.812
C03404=1017.687,253.968,-133.139,169.139,51.356,159.812
C03405=1017.692,254.216,-133.167,169.143,51.349,159.811
C03406=1017.699,254.464,-133.195,169.148,51.343,159.810
C03407=1017.704,254.712,-133.223,169.153,51.337,159.810
C03408=1017.711,254.961,-133.250,169.157,51.331,159.809
C03409=1017.717,255.209,-133.279,169.162,51.325,159.809
C03410=1017.722,255.457,-133.307,169.166,51.318,159.808
C03411=1017.729,255.706,-133.334,169.171,51.312,159.808
C03412=1017.735,255.955,-133.363,169.176,51.306,159.807
C03413=1017.740,256.203,-133.391,169.181,51.300,159.807
C03414=1017.747,256.450,-133.419,169.186,51.294,159.807
C03415=1017.753,256.699,-133.447,169.189,51.288,159.806
C03416=1017.758,256.947,-133.475,169.194,51.282,159.805
C03417=1017.765,257.196,-133.503,169.199,51.275,159.805
C03418=1017.771,257.444,-133.531,169.204,51.270,159.804
C03419=1017.777,257.692,-133.559,169.208,51.263,159.804
C03420=1017.783,257.941,-133.587,169.214,51.257,159.803
C03421=1017.789,258.189,-133.616,169.218,51.251,159.803
C03422=1017.796,258.438,-133.644,169.222,51.245,159.802
C03423=1017.801,258.686,-133.672,169.227,51.240,159.802
C03424=1017.807,258.934,-133.700,169.232,51.233,159.801
C03425=1017.814,259.183,-133.728,169.237,51.227,159.801
C03426=1017.820,259.431,-133.757,169.241,51.221,159.800
C03427=1017.826,259.679,-133.785,169.247,51.215,159.800
C03428=1017.832,259.927,-133.813,169.251,51.210,159.800
C03429=1017.839,260.176,-133.842,169.256,51.204,159.799
C03430=1017.844,260.425,-133.871,169.260,51.197,159.799
C03431=1017.849,260.672,-133.899,169.265,51.191,159.798
C03432=1017.855,260.921,-133.928,169.269,51.186,159.798
C03433=1017.862,261.169,-133.957,169.274,51.180,159.797
C03434=1017.868,261.418,-133.985,169.279,51.174,159.797
C03435=1017.873,261.665,-134.014,169.284,51.169,159.797
C03436=1017.879,261.914,-134.042,169.288,51.163,159.796
C03437=1017.885,262.162,-134.071,169.293,51.157,159.796
C03438=1017.891,262.411,-134.099,169.298,51.151,159.795
C03439=1017.898,262.659,-134.128,169.302,51.146,159.795
C03440=1017.902,262.887,-134.155,169.308,51.140,159.794
C03441=1017.908,263.116,-134.181,169.312,51.135,159.794
C03442=1017.914,263.344,-134.208,169.316,51.130,159.794
C03443=1017.919,263.572,-134.234,169.320,51.125,159.793
C03444=1017.925,263.801,-134.260,169.324,51.119,159.793
C03445=1017.930,264.030,-134.287,169.329,51.114,159.792
C03446=1017.936,264.258,-134.314,169.334,51.109,159.792
C03447=1017.941,264.487,-134.340,169.338,51.103,159.792
C03448=1017.947,264.735,-134.369,169.343,51.098,159.791
C03449=1017.953,264.984,-134.398,169.348,51.092,159.791
C03450=1017.960,265.232,-134.427,169.352,51.086,159.790
C03451=1017.965,265.479,-134.455,169.357,51.081,159.790
C03452=1017.972,265.727,-134.484,169.362,51.075,159.790
C03453=1017.977,265.976,-134.514,169.366,51.070,159.789
C03454=1017.983,266.225,-134.542,169.371,51.064,159.789
C03455=1017.989,266.473,-134.571,169.376,51.059,159.789
C03456=1017.996,266.721,-134.600,169.380,51.053,159.788
C03457=1018.002,266.969,-134.630,169.386,51.047,159.788
C03458=1018.007,267.218,-134.659,169.391,51.042,159.788
C03459=1018.014,267.466,-134.688,169.396,51.036,159.787
C03460=1018.020,267.714,-134.717,169.400,51.031,159.787
C03461=1018.026,267.962,-134.746,169.405,51.025,159.786
C03462=1018.031,268.211,-134.775,169.411,51.020,159.786
C03463=1018.037,268.459,-134.804,169.415,51.015,159.786
C03464=1018.044,268.707,-134.833,169.420,51.009,159.785
C03465=1018.050,268.955,-134.862,169.425,51.003,159.785
C03466=1018.055,269.203,-134.892,169.429,50.998,159.785
C03467=1018.061,269.451,-134.921,169.434,50.993,159.784
C03468=1018.068,269.699,-134.950,169.439,50.987,159.784
C03469=1018.073,269.947,-134.980,169.444,50.982,159.783
C03470=1018.079,270.195,-135.009,169.449,50.976,159.783
C03471=1018.085,270.444,-135.039,169.454,50.971,159.783
C03472=1018.092,270.693,-135.068,169.458,50.966,159.782
C03473=1018.098,270.941,-135.097,169.463,50.960,159.782
C03474=1018.104,271.189,-135.127,169.469,50.955,159.782
C03475=1018.110,271.437,-135.157,169.473,50.950,159.781
C03476=1018.116,271.685,-135.186,169.478,50.945,159.781
C03477=1018.122,271.933,-135.215,169.483,50.939,159.781
C03478=1018.128,272.181,-135.244,169.488,50.934,159.781
C03479=1018.134,272.430,-135.274,169.493,50.928,159.780
C03480=1018.140,272.677,-135.304,169.497,50.924,159.780
C03481=1018.146,272.926,-135.333,169.502,50.918,159.779
C03482=1018.152,273.174,-135.362,169.508,50.913,159.779
C03483=1018.158,273.422,-135.393,169.512,50.908,159.779
C03484=1018.164,273.670,-135.422,169.517,50.902,159.779
C03485=1018.170,273.918,-135.451,169.523,50.897,159.778
C03486=1018.177,274.167,-135.481,169.527,50.892,159.778
C03487=1018.182,274.415,-135.511,169.532,50.887,159.778
C03488=1018.188,274.663,-135.540,169.538,50.882,159.778
C03489=1018.194,274.911,-135.570,169.542,50.876,159.777
C03490=1018.201,275.159,-135.600,169.547,50.871,159.777
C03491=1018.206,275.407,-135.630,169.552,50.866,159.777
C03492=1018.213,275.656,-135.659,169.557,50.861,159.776
C03493=1018.219,275.904,-135.690,169.562,50.856,159.776
C03494=1018.225,276.152,-135.719,169.567,50.851,159.776
C03495=1018.231,276.399,-135.749,169.572,50.846,159.776
C03496=1018.237,276.648,-135.778,169.577,50.840,159.775
C03497=1018.244,276.896,-135.809,169.582,50.835,159.775
C03498=1018.249,277.145,-135.838,169.587,50.830,159.775
C03499=1018.255,277.392,-135.869,169.592,50.826,159.774
C03500=1018.261,277.623,-135.897,169.597,50.820,159.774
C03501=1018.267,277.854,-135.924,169.602,50.816,159.774
C03502=1018.272,278.085,-135.953,169.606,50.811,159.774
C03503=1018.278,278.316,-135.981,169.611,50.807,159.774
C03504=1018.284,278.546,-136.008,169.615,50.802,159.773
C03505=1018.289,278.777,-136.037,169.620,50.798,159.773
C03506=1018.295,279.007,-136.065,169.624,50.793,159.773
C03507=1018.300,279.239,-136.092,169.629,50.789,159.773
C03508=1018.306,279.486,-136.122,169.635,50.784,159.773
C03509=1018.313,279.735,-136.153,169.640,50.779,159.772
C03510=1018.319,279.983,-136.183,169.645,50.774,159.772
C03511=1018.325,280.230,-136.213,169.650,50.769,159.772
C03512=1018.331,280.479,-136.243,169.655,50.764,159.772
C03513=1018.337,280.727,-136.273,169.660,50.759,159.771
C03514=1018.343,280.975,-136.304,169.666,50.754,159.771
C03515=1018.350,281.223,-136.334,169.670,50.749,159.771
C03516=1018.356,281.471,-136.364,169.675,50.744,159.771
C03517=1018.362,281.719,-136.394,169.680,50.740,159.770
C03518=1018.368,281.967,-136.425,169.685,50.734,159.770
C03519=1018.375,282.215,-136.455,169.691,50.729,159.770
C03520=1018.381,282.464,-136.485,169.695,50.725,159.770
C03521=1018.387,282.712,-136.515,169.701,50.720,159.770
C03522=1018.392,282.960,-136.546,169.705,50.715,159.769
C03523=1018.399,283.208,-136.576,169.711,50.711,159.769
C03524=1018.405,283.456,-136.606,169.717,50.706,159.769
C03525=1018.412,283.704,-136.637,169.721,50.701,159.769
C03526=1018.418,283.952,-136.667,169.727,50.696,159.769
C03527=1018.423,284.200,-136.698,169.731,50.691,159.768
C03528=1018.431,284.448,-136.728,169.737,50.687,159.768
C03529=1018.437,284.695,-136.759,169.742,50.682,159.768
C03530=1018.443,284.944,-136.789,169.747,50.677,159.768
C03531=1018.449,285.192,-136.820,169.752,50.672,159.768
C03532=1018.455,285.440,-136.850,169.757,50.668,159.768
C03533=1018.461,285.688,-136.881,169.763,50.663,159.767
C03534=1018.468,285.937,-136.912,169.768,50.659,159.767
C03535=1018.474,286.184,-136.943,169.773,50.654,159.767
C03536=1018.480,286.432,-136.973,169.779,50.649,159.767
C03537=1018.486,286.680,-137.004,169.783,50.645,159.767
C03538=1018.493,286.928,-137.035,169.789,50.640,159.767
C03539=1018.498,287.176,-137.065,169.794,50.636,159.767
C03540=1018.505,287.424,-137.096,169.799,50.630,159.766
C03541=1018.511,287.672,-137.127,169.804,50.626,159.766
C03542=1018.517,287.920,-137.158,169.810,50.621,159.766
C03543=1018.523,288.168,-137.188,169.815,50.617,159.766
C03544=1018.530,288.416,-137.220,169.820,50.612,159.766
C03545=1018.536,288.664,-137.250,169.826,50.608,159.766
C03546=1018.542,288.912,-137.281,169.830,50.603,159.766
C03547=1018.549,289.160,-137.312,169.836,50.599,159.766
C03548=1018.555,289.408,-137.343,169.841,50.594,159.765
C03549=1018.561,289.656,-137.375,169.847,50.590,159.765
C03550=1018.567,289.904,-137.405,169.851,50.586,159.765
C03551=1018.573,290.152,-137.436,169.857,50.581,159.765
C03552=1018.580,290.400,-137.467,169.863,50.576,159.765
C03553=1018.586,290.648,-137.498,169.867,50.572,159.765
C03554=1018.593,290.895,-137.530,169.873,50.567,159.765
C03555=1018.598,291.143,-137.560,169.878,50.563,159.765
C03556=1018.605,291.391,-137.591,169.883,50.558,159.764
C03557=1018.611,291.640,-137.622,169.888,50.554,159.764
C03558=1018.617,291.887,-137.654,169.894,50.550,159.764
C03559=1018.624,292.135,-137.685,169.899,50.546,159.764
C03560=1018.629,292.372,-137.715,169.905,50.541,159.764
C03561=1018.636,292.609,-137.745,169.910,50.537,159.764
C03562=1018.641,292.846,-137.774,169.915,50.533,159.764
C03563=1018.648,293.083,-137.804,169.920,50.528,159.764
C03564=1018.654,293.320,-137.835,169.925,50.525,159.764
C03565=1018.659,293.557,-137.864,169.930,50.521,159.764
C03566=1018.665,293.793,-137.894,169.935,50.517,159.764
C03567=1018.671,294.031,-137.925,169.940,50.513,159.764
C03568=1018.677,294.278,-137.957,169.946,50.509,159.764
C03569=1018.684,294.526,-137.988,169.951,50.505,159.764
C03570=1018.690,294.774,-138.020,169.957,50.500,159.764
C03571=1018.696,295.022,-138.052,169.962,50.496,159.764
C03572=1018.702,295.270,-138.084,169.967,50.492,159.764
C03573=1018.708,295.518,-138.115,169.972,50.488,159.764
C03574=1018.714,295.766,-138.147,169.978,50.483,159.764
C03575=1018.721,296.013,-138.178,169.983,50.479,159.764
C03576=1018.727,296.261,-138.210,169.989,50.475,159.764
C03577=1018.732,296.510,-138.242,169.994,50.471,159.763
C03578=1018.739,296.758,-138.274,170.000,50.467,159.764
